C05489=1180.619,-50.249,-42.680,179.529,5.743,149.159
C05490=1180.625,-50.498,-42.668,179.526,5.742,149.160
C05491=1180.631,-50.748,-42.656,179.523,5.742,149.160
C05492=1180.635,-50.998,-42.645,179.521,5.741,149.161
C05493=1180.641,-51.248,-42.633,179.519,5.741,149.162
C05494=1180.645,-51.497,-42.622,179.516,5.741,149.162
C05495=1180.651,-51.747,-42.610,179.514,5.740,149.163
C05496=1180.656,-51.996,-42.599,179.512,5.740,149.163
C05497=1180.662,-52.246,-42.587,179.509,5.740,149.164
C05498=1180.666,-52.496,-42.576,179.507,5.739,149.165
C05499=1180.672,-52.746,-42.565,179.505,5.739,149.165
C05500=1180.677,-52.995,-42.554,179.502,5.738,149.166
C05501=1180.683,-53.245,-42.542,179.500,5.738,149.166
C05502=1180.687,-53.495,-42.531,179.498,5.738,149.167
C05503=1180.693,-53.745,-42.519,179.495,5.737,149.168
C05504=1180.697,-53.994,-42.507,179.493,5.737,149.168
C05505=1180.704,-54.244,-42.496,179.491,5.737,149.169
C05506=1180.708,-54.493,-42.485,179.488,5.737,149.170
C05507=1180.714,-54.743,-42.473,179.486,5.736,149.170
C05508=1180.718,-54.993,-42.461,179.483,5.735,149.171
C05509=1180.723,-55.243,-42.451,179.481,5.736,149.172
C05510=1180.729,-55.492,-42.439,179.479,5.735,149.172
C05511=1180.734,-55.742,-42.428,179.476,5.734,149.173
C05512=1180.739,-55.992,-42.416,179.474,5.735,149.174
C05513=1180.744,-56.242,-42.405,179.472,5.734,149.174
C05514=1180.750,-56.491,-42.393,179.469,5.734,149.175
C05515=1180.755,-56.740,-42.382,179.467,5.733,149.175
C05516=1180.760,-56.991,-42.372,179.465,5.733,149.176
C05517=1180.765,-57.241,-42.360,179.462,5.733,149.177
C05518=1180.771,-57.489,-42.349,179.460,5.732,149.177
C05519=1180.776,-57.739,-42.337,179.458,5.732,149.178
C05520=1180.781,-57.989,-42.326,179.456,5.732,149.179
C05521=1180.786,-58.239,-42.315,179.453,5.731,149.179
C05522=1180.792,-58.489,-42.303,179.451,5.731,149.180
C05523=1180.796,-58.738,-42.292,179.449,5.731,149.180
C05524=1180.802,-58.988,-42.280,179.446,5.731,149.181
C05525=1180.807,-59.238,-42.270,179.444,5.730,149.182
C05526=1180.812,-59.487,-42.259,179.442,5.730,149.182
C05527=1180.818,-59.737,-42.247,179.439,5.730,149.183
C05528=1180.822,-59.987,-42.236,179.437,5.729,149.183
C05529=1180.828,-60.236,-42.225,179.434,5.729,149.184
C05530=1180.833,-60.486,-42.213,179.432,5.729,149.185
C05531=1180.838,-60.736,-42.202,179.430,5.728,149.185
C05532=1180.844,-60.985,-42.192,179.427,5.728,149.186
C05533=1180.849,-61.235,-42.180,179.425,5.728,149.187
C05534=1180.854,-61.485,-42.169,179.423,5.727,149.187
C05535=1180.859,-61.735,-42.159,179.420,5.727,149.188
C05536=1180.865,-61.985,-42.147,179.418,5.727,149.189
C05537=1180.869,-62.234,-42.135,179.416,5.726,149.189
C05538=1180.875,-62.484,-42.125,179.413,5.726,149.190
C05539=1180.880,-62.734,-42.113,179.411,5.725,149.190
C05540=1180.885,-62.983,-42.102,179.409,5.726,149.191
C05541=1180.891,-63.233,-42.092,179.406,5.725,149.192
C05542=1180.895,-63.482,-42.081,179.404,5.724,149.192
C05543=1180.901,-63.732,-42.069,179.402,5.725,149.193
C05544=1180.906,-63.982,-42.058,179.399,5.724,149.194
C05545=1180.911,-64.232,-42.047,179.397,5.723,149.194
C05546=1180.916,-64.482,-42.037,179.395,5.724,149.195
C05547=1180.922,-64.731,-42.025,179.393,5.723,149.196
C05548=1180.927,-64.981,-42.014,179.390,5.723,149.196
C05549=1180.933,-65.230,-42.004,179.388,5.723,149.197
C05550=1180.937,-65.480,-41.992,179.386,5.723,149.197
C05551=1180.943,-65.730,-41.981,179.383,5.722,149.198
C05552=1180.948,-65.979,-41.970,179.381,5.722,149.199
C05553=1180.953,-66.230,-41.960,179.379,5.722,149.199
C05554=1180.959,-66.478,-41.949,179.376,5.721,149.200
C05555=1180.964,-66.729,-41.938,179.374,5.721,149.200
C05556=1180.969,-66.979,-41.926,179.372,5.721,149.201
C05557=1180.974,-67.228,-41.915,179.370,5.720,149.202
C05558=1180.979,-67.478,-41.905,179.367,5.720,149.202
C05559=1180.985,-67.727,-41.894,179.365,5.720,149.203
C05560=1180.990,-67.977,-41.883,179.363,5.719,149.204
C05561=1180.995,-68.227,-41.871,179.360,5.719,149.204
C05562=1181.001,-68.476,-41.861,179.358,5.719,149.205
C05563=1181.006,-68.727,-41.851,179.356,5.718,149.205
C05564=1181.011,-68.976,-41.840,179.353,5.718,149.206
C05565=1181.017,-69.226,-41.828,179.351,5.718,149.207
C05566=1181.022,-69.475,-41.818,179.349,5.718,149.207
C05567=1181.027,-69.725,-41.807,179.346,5.717,149.208
C05568=1181.032,-69.975,-41.796,179.344,5.717,149.209
C05569=1181.037,-70.225,-41.785,179.342,5.717,149.209
C05570=1181.042,-70.474,-41.774,179.340,5.716,149.210
C05571=1181.047,-70.724,-41.764,179.338,5.716,149.210
C05572=1181.053,-70.974,-41.753,179.335,5.716,149.211
C05573=1181.058,-71.223,-41.742,179.333,5.715,149.212
C05574=1181.063,-71.473,-41.731,179.331,5.716,149.212
C05575=1181.069,-71.722,-41.720,179.328,5.715,149.213
C05576=1181.074,-71.973,-41.710,179.326,5.714,149.214
C05577=1181.079,-72.222,-41.700,179.324,5.715,149.214
C05578=1181.084,-72.472,-41.688,179.321,5.714,149.215
C05579=1181.090,-72.721,-41.678,179.319,5.714,149.215
C05580=1181.095,-72.972,-41.668,179.317,5.714,149.216
C05581=1181.101,-73.221,-41.656,179.315,5.713,149.217
C05582=1181.106,-73.471,-41.645,179.312,5.713,149.217
C05583=1181.111,-73.721,-41.635,179.310,5.713,149.218
C05584=1181.116,-73.970,-41.624,179.308,5.712,149.218
C05585=1181.122,-74.220,-41.614,179.306,5.713,149.219
C05586=1181.127,-74.470,-41.603,179.303,5.712,149.220
C05587=1181.132,-74.719,-41.592,179.301,5.711,149.220
C05588=1181.137,-74.969,-41.582,179.299,5.712,149.221
C05589=1181.142,-75.219,-41.571,179.296,5.711,149.222
C05590=1181.148,-75.490,-41.559,179.294,5.711,149.222
C05591=1181.153,-75.761,-41.548,179.291,5.710,149.223
C05592=1181.159,-76.031,-41.536,179.289,5.711,149.224
C05593=1181.165,-76.303,-41.525,179.286,5.710,149.224
C05594=1181.170,-76.553,-41.514,179.284,5.709,149.225
C05595=1181.176,-76.803,-41.504,179.282,5.710,149.226
C05596=1181.181,-77.052,-41.493,179.279,5.709,149.226
C05597=1181.186,-77.302,-41.483,179.277,5.709,149.227
C05598=1181.192,-77.551,-41.472,179.275,5.709,149.227
C05599=1181.197,-77.802,-41.462,179.273,5.708,149.228
C05600=1181.202,-78.051,-41.451,179.270,5.708,149.229
C05601=1181.207,-78.301,-41.440,179.268,5.708,149.229
C05602=1181.213,-78.550,-41.430,179.266,5.707,149.230
C05603=1181.218,-78.801,-41.419,179.263,5.707,149.231
C05604=1181.223,-79.050,-41.409,179.262,5.707,149.231
C05605=1181.229,-79.299,-41.398,179.259,5.707,149.232
C05606=1181.234,-79.549,-41.388,179.257,5.707,149.232
C05607=1181.239,-79.798,-41.378,179.255,5.706,149.233
C05608=1181.244,-80.049,-41.368,179.252,5.706,149.234
C05609=1181.249,-80.298,-41.357,179.251,5.706,149.234
C05610=1181.255,-80.548,-41.347,179.248,5.705,149.235
C05611=1181.260,-80.798,-41.337,179.245,5.705,149.236
C05612=1181.265,-81.047,-41.326,179.244,5.705,149.236
C05613=1181.270,-81.297,-41.315,179.241,5.705,149.237
C05614=1181.276,-81.547,-41.305,179.239,5.705,149.237
C05615=1181.281,-81.797,-41.294,179.237,5.704,149.238
C05616=1181.286,-82.047,-41.284,179.234,5.704,149.239
C05617=1181.292,-82.296,-41.274,179.232,5.704,149.239
C05618=1181.297,-82.546,-41.263,179.230,5.703,149.240
C05619=1181.302,-82.796,-41.254,179.227,5.703,149.241
C05620=1181.307,-83.045,-41.243,179.225,5.703,149.241
C05621=1181.312,-83.295,-41.233,179.223,5.703,149.242
C05622=1181.318,-83.545,-41.223,179.221,5.703,149.242
C05623=1181.323,-83.795,-41.211,179.218,5.702,149.243
C05624=1181.328,-84.044,-41.201,179.216,5.702,149.244
C05625=1181.334,-84.294,-41.191,179.214,5.702,149.244
C05626=1181.339,-84.544,-41.180,179.212,5.701,149.245
C05627=1181.344,-84.793,-41.171,179.210,5.701,149.245
C05628=1181.349,-85.043,-41.161,179.207,5.701,149.246
C05629=1181.354,-85.293,-41.150,179.205,5.700,149.247
C05630=1181.360,-85.542,-41.140,179.203,5.701,149.247
C05631=1181.365,-85.792,-41.130,179.200,5.700,149.248
C05632=1181.370,-86.042,-41.119,179.199,5.700,149.248
C05633=1181.375,-86.291,-41.109,179.196,5.700,149.249
C05634=1181.381,-86.541,-41.099,179.194,5.699,149.250
C05635=1181.386,-86.791,-41.089,179.192,5.699,149.250
C05636=1181.391,-87.041,-41.078,179.189,5.699,149.251
C05637=1181.397,-87.290,-41.068,179.188,5.699,149.252
C05638=1181.402,-87.541,-41.059,179.185,5.699,149.252
C05639=1181.407,-87.790,-41.049,179.183,5.698,149.253
C05640=1181.413,-88.040,-41.039,179.181,5.698,149.253
C05641=1181.418,-88.290,-41.028,179.178,5.698,149.254
C05642=1181.423,-88.539,-41.018,179.176,5.698,149.255
C05643=1181.428,-88.789,-41.008,179.174,5.697,149.255
C05644=1181.433,-89.039,-40.998,179.171,5.697,149.256
C05645=1181.439,-89.289,-40.987,179.169,5.697,149.257
C05646=1181.444,-89.538,-40.977,179.167,5.696,149.257
C05647=1181.449,-89.788,-40.967,179.165,5.697,149.258
C05648=1181.454,-90.038,-40.957,179.162,5.696,149.258
C05649=1181.460,-90.288,-40.947,179.160,5.695,149.259
C05650=1181.465,-90.537,-40.938,179.158,5.696,149.260
C05651=1181.470,-90.787,-40.927,179.156,5.695,149.260
C05652=1181.476,-91.037,-40.917,179.154,5.695,149.261
C05653=1181.481,-91.287,-40.907,179.152,5.695,149.261
C05654=1181.486,-91.536,-40.897,179.149,5.694,149.262
C05655=1181.491,-91.786,-40.887,179.147,5.695,149.263
C05656=1181.497,-92.036,-40.877,179.145,5.694,149.263
C05657=1181.503,-92.286,-40.867,179.143,5.694,149.264
C05658=1181.507,-92.536,-40.857,179.140,5.693,149.264
C05659=1181.512,-92.785,-40.847,179.138,5.693,149.265
C05660=1181.518,-93.035,-40.837,179.136,5.693,149.266
C05661=1181.523,-93.285,-40.828,179.134,5.693,149.266
C05662=1181.528,-93.535,-40.817,179.131,5.693,149.267
C05663=1181.534,-93.784,-40.807,179.129,5.692,149.267
C05664=1181.539,-94.034,-40.797,179.127,5.693,149.268
C05665=1181.545,-94.284,-40.788,179.125,5.692,149.269
C05666=1181.550,-94.533,-40.778,179.122,5.691,149.269
C05667=1181.554,-94.783,-40.768,179.121,5.691,149.270
C05668=1181.560,-95.033,-40.757,179.118,5.691,149.271
C05669=1181.566,-95.283,-40.748,179.116,5.691,149.271
C05670=1181.571,-95.532,-40.738,179.114,5.691,149.272
C05671=1181.576,-95.782,-40.728,179.112,5.691,149.272
C05672=1181.581,-96.032,-40.718,179.109,5.690,149.273
C05673=1181.587,-96.282,-40.709,179.107,5.690,149.274
C05674=1181.592,-96.531,-40.698,179.105,5.690,149.274
C05675=1181.597,-96.781,-40.689,179.103,5.689,149.275
C05676=1181.603,-97.031,-40.679,179.101,5.689,149.275
C05677=1181.608,-97.281,-40.669,179.098,5.689,149.276
C05678=1181.613,-97.530,-40.659,179.097,5.689,149.277
C05679=1181.619,-97.780,-40.650,179.094,5.689,149.277
C05680=1181.624,-98.030,-40.640,179.091,5.688,149.278
C05681=1181.629,-98.279,-40.630,179.090,5.688,149.278
C05682=1181.634,-98.530,-40.620,179.087,5.688,149.279
C05683=1181.639,-98.779,-40.610,179.085,5.688,149.280
C05684=1181.645,-99.029,-40.600,179.083,5.688,149.280
C05685=1181.650,-99.279,-40.591,179.081,5.688,149.281
C05686=1181.656,-99.528,-40.581,179.078,5.687,149.282
C05687=1181.661,-99.777,-40.571,179.077,5.687,149.282
C05688=1181.666,-100.028,-40.562,179.074,5.687,149.283
C05689=1181.671,-100.278,-40.551,179.072,5.686,149.283
C05690=1181.677,-100.528,-40.542,179.070,5.686,149.284
C05691=1181.682,-100.777,-40.532,179.067,5.686,149.285
C05692=1181.687,-101.026,-40.523,179.066,5.686,149.285
C05693=1181.693,-101.277,-40.513,179.063,5.686,149.286
C05694=1181.698,-101.549,-40.503,179.061,5.686,149.286
C05695=1181.704,-101.820,-40.492,179.059,5.685,149.287
C05696=1181.709,-102.092,-40.482,179.056,5.685,149.288
C05697=1181.716,-102.363,-40.471,179.053,5.684,149.289
C05698=1181.721,-102.613,-40.462,179.052,5.685,149.289
C05699=1181.726,-102.863,-40.452,179.049,5.684,149.290
C05700=1181.731,-103.113,-40.442,179.047,5.684,149.290
C05701=1181.737,-103.363,-40.433,179.045,5.684,149.291
C05702=1181.742,-103.612,-40.423,179.043,5.684,149.291
C05703=1181.748,-103.862,-40.414,179.041,5.683,149.292
C05704=1181.753,-104.111,-40.404,179.039,5.683,149.293
C05705=1181.758,-104.362,-40.394,179.036,5.683,149.293
C05706=1181.763,-104.611,-40.385,179.035,5.683,149.294
C05707=1181.768,-104.861,-40.376,179.032,5.683,149.295
C05708=1181.773,-105.111,-40.365,179.030,5.682,149.295
C05709=1181.779,-105.361,-40.356,179.028,5.682,149.296
C05710=1181.784,-105.610,-40.346,179.026,5.681,149.296
C05711=1181.789,-105.860,-40.337,179.023,5.682,149.297
C05712=1181.795,-106.110,-40.327,179.021,5.681,149.298
C05713=1181.800,-106.360,-40.318,179.019,5.681,149.298
C05714=1181.806,-106.610,-40.309,179.016,5.681,149.299
C05715=1181.811,-106.859,-40.299,179.015,5.681,149.299
C05716=1181.816,-107.109,-40.290,179.012,5.681,149.300
C05717=1181.822,-107.358,-40.280,179.011,5.681,149.300
C05718=1181.827,-107.608,-40.271,179.008,5.680,149.301
C05719=1181.832,-107.858,-40.261,179.006,5.680,149.302
C05720=1181.838,-108.108,-40.252,179.004,5.680,149.302
C05721=1181.843,-108.357,-40.243,179.002,5.680,149.303
C05722=1181.848,-108.607,-40.233,178.999,5.680,149.304
C05723=1181.853,-108.858,-40.224,178.997,5.679,149.304
C05724=1181.859,-109.108,-40.214,178.995,5.679,149.305
C05725=1181.864,-109.357,-40.205,178.993,5.678,149.305
C05726=1181.869,-109.607,-40.196,178.991,5.679,149.306
C05727=1181.874,-109.856,-40.185,178.989,5.678,149.306
C05728=1181.880,-110.106,-40.177,178.987,5.678,149.307
C05729=1181.885,-110.356,-40.168,178.984,5.678,149.308
C05730=1181.890,-110.606,-40.157,178.982,5.678,149.308
C05731=1181.896,-110.855,-40.149,178.980,5.677,149.309
C05732=1181.901,-111.105,-40.140,178.978,5.678,149.310
C05733=1181.906,-111.355,-40.129,178.976,5.677,149.310
C05734=1181.912,-111.605,-40.121,178.974,5.677,149.311
C05735=1181.917,-111.855,-40.112,178.972,5.677,149.311
C05736=1181.923,-112.105,-40.102,178.969,5.677,149.312
C05737=1181.927,-112.354,-40.093,178.967,5.676,149.312
C05738=1181.933,-112.604,-40.084,178.965,5.677,149.313
C05739=1181.939,-112.854,-40.074,178.963,5.676,149.314
C05740=1181.944,-113.104,-40.065,178.961,5.676,149.314
C05741=1181.949,-113.353,-40.056,178.959,5.676,149.315
C05742=1181.954,-113.603,-40.046,178.957,5.676,149.316
C05743=1181.960,-113.853,-40.037,178.954,5.675,149.316
C05744=1181.965,-114.103,-40.028,178.953,5.675,149.317
C05745=1181.970,-114.352,-40.019,178.950,5.675,149.317
C05746=1181.976,-114.602,-40.010,178.949,5.675,149.318
C05747=1181.981,-114.851,-40.001,178.946,5.674,149.318
C05748=1181.986,-115.101,-39.992,178.944,5.674,149.319
C05749=1181.992,-115.351,-39.982,178.942,5.674,149.320
C05750=1181.997,-115.601,-39.973,178.939,5.673,149.320
C05751=1182.002,-115.851,-39.964,178.937,5.674,149.321
C05752=1182.008,-116.100,-39.955,178.935,5.673,149.321
C05753=1182.013,-116.351,-39.945,178.933,5.673,149.322
C05754=1182.019,-116.600,-39.937,178.931,5.673,149.323
C05755=1182.024,-116.850,-39.927,178.929,5.673,149.323
C05756=1182.029,-117.099,-39.918,178.927,5.672,149.324
C05757=1182.034,-117.349,-39.909,178.924,5.673,149.324
C05758=1182.040,-117.599,-39.900,178.922,5.672,149.325
C05759=1182.045,-117.849,-39.891,178.920,5.672,149.326
C05760=1182.050,-118.099,-39.882,178.918,5.671,149.326
C05761=1182.055,-118.348,-39.872,178.916,5.671,149.327
C05762=1182.061,-118.598,-39.864,178.914,5.671,149.327
C05763=1182.067,-118.848,-39.854,178.912,5.671,149.328
C05764=1182.072,-119.098,-39.845,178.909,5.671,149.329
C05765=1182.077,-119.347,-39.836,178.908,5.671,149.329
C05766=1182.082,-119.597,-39.828,178.905,5.670,149.330
C05767=1182.087,-119.847,-39.819,178.904,5.670,149.330
C05768=1182.093,-120.097,-39.809,178.901,5.670,149.331
C05769=1182.098,-120.347,-39.800,178.899,5.670,149.331
C05770=1182.104,-120.597,-39.791,178.897,5.670,149.332
C05771=1182.109,-120.847,-39.782,178.895,5.670,149.333
C05772=1182.114,-121.095,-39.773,178.893,5.669,149.333
C05773=1182.119,-121.345,-39.764,178.891,5.669,149.334
C05774=1182.124,-121.595,-39.755,178.889,5.669,149.334
C05775=1182.130,-121.845,-39.746,178.886,5.669,149.335
C05776=1182.136,-122.095,-39.737,178.885,5.669,149.336
C05777=1182.141,-122.345,-39.728,178.882,5.669,149.336
C05778=1182.146,-122.595,-39.719,178.881,5.669,149.337
C05779=1182.151,-122.845,-39.710,178.878,5.668,149.337
C05780=1182.157,-123.094,-39.702,178.876,5.668,149.338
C05781=1182.162,-123.344,-39.693,178.874,5.668,149.338
C05782=1182.167,-123.593,-39.684,178.872,5.668,149.339
C05783=1182.173,-123.844,-39.674,178.870,5.667,149.340
C05784=1182.178,-124.094,-39.666,178.868,5.668,149.340
C05785=1182.183,-124.343,-39.657,178.866,5.667,149.341
C05786=1182.189,-124.593,-39.648,178.863,5.667,149.342
C05787=1182.194,-124.842,-39.639,178.861,5.666,149.342
C05788=1182.199,-125.092,-39.630,178.860,5.666,149.343
C05789=1182.205,-125.342,-39.621,178.857,5.666,149.343
C05790=1182.210,-125.593,-39.613,178.855,5.666,149.344
C05791=1182.215,-125.842,-39.604,178.853,5.666,149.344
C05792=1182.220,-126.092,-39.595,178.851,5.666,149.345
C05793=1182.226,-126.341,-39.587,178.848,5.665,149.346
C05794=1182.231,-126.591,-39.578,178.847,5.665,149.346
C05795=1182.237,-126.841,-39.569,178.845,5.665,149.347
C05796=1182.242,-127.091,-39.560,178.843,5.665,149.347
C05797=1182.248,-127.341,-39.551,178.840,5.664,149.348
C05798=1181.827,-127.352,-39.591,178.837,5.668,149.350
C05799=1181.821,-127.102,-39.600,178.839,5.668,149.349
C05800=1181.816,-126.853,-39.609,178.841,5.669,149.349
C05801=1181.810,-126.603,-39.618,178.843,5.669,149.348
C05802=1181.805,-126.353,-39.626,178.845,5.669,149.348
C05803=1181.800,-126.103,-39.635,178.847,5.669,149.347
C05804=1181.794,-125.852,-39.644,178.849,5.669,149.346
C05805=1181.789,-125.602,-39.653,178.852,5.669,149.346
C05806=1181.783,-125.353,-39.662,178.853,5.669,149.345
C05807=1181.778,-125.103,-39.670,178.855,5.670,149.345
C05808=1181.773,-124.854,-39.679,178.857,5.670,149.344
C05809=1181.767,-124.604,-39.688,178.860,5.670,149.343
C05810=1181.762,-124.354,-39.697,178.862,5.670,149.343
C05811=1181.757,-124.104,-39.706,178.864,5.671,149.342
C05812=1181.751,-123.855,-39.715,178.866,5.670,149.342
C05813=1181.746,-123.605,-39.723,178.868,5.671,149.341
C05814=1181.741,-123.355,-39.732,178.870,5.671,149.341
C05815=1181.736,-123.105,-39.741,178.872,5.671,149.340
C05816=1181.730,-122.855,-39.751,178.874,5.671,149.339
C05817=1181.725,-122.605,-39.760,178.877,5.672,149.339
C05818=1181.720,-122.356,-39.769,178.878,5.672,149.338
C05819=1181.714,-122.106,-39.777,178.881,5.672,149.337
C05820=1181.709,-121.857,-39.786,178.883,5.672,149.337
C05821=1181.704,-121.607,-39.795,178.885,5.673,149.336
C05822=1181.698,-121.357,-39.804,178.887,5.673,149.336
C05823=1181.693,-121.107,-39.813,178.889,5.673,149.335
C05824=1181.687,-120.857,-39.822,178.891,5.673,149.335
C05825=1181.682,-120.607,-39.831,178.893,5.674,149.334
C05826=1181.677,-120.357,-39.840,178.895,5.673,149.333
C05827=1181.671,-120.108,-39.848,178.898,5.674,149.333
C05828=1181.666,-119.859,-39.858,178.900,5.674,149.332
C05829=1181.661,-119.609,-39.867,178.902,5.674,149.332
C05830=1181.655,-119.359,-39.876,178.903,5.674,149.331
C05831=1181.650,-119.109,-39.885,178.906,5.675,149.330
C05832=1181.645,-118.859,-39.894,178.908,5.675,149.330
C05833=1181.640,-118.609,-39.903,178.910,5.675,149.329
C05834=1181.635,-118.359,-39.912,178.912,5.675,149.329
C05835=1181.629,-118.109,-39.922,178.915,5.675,149.328
C05836=1181.623,-117.859,-39.930,178.916,5.675,149.328
C05837=1181.619,-117.610,-39.940,178.919,5.676,149.327
C05838=1181.613,-117.361,-39.949,178.921,5.676,149.326
C05839=1181.608,-117.111,-39.957,178.923,5.676,149.326
C05840=1181.602,-116.861,-39.967,178.925,5.676,149.325
C05841=1181.597,-116.611,-39.976,178.928,5.677,149.324
C05842=1181.591,-116.361,-39.985,178.929,5.677,149.324
C05843=1181.587,-116.112,-39.994,178.931,5.677,149.323
C05844=1181.581,-115.862,-40.004,178.933,5.677,149.323
C05845=1181.576,-115.612,-40.013,178.936,5.678,149.322
C05846=1181.570,-115.362,-40.022,178.938,5.677,149.322
C05847=1181.565,-115.112,-40.031,178.940,5.678,149.321
C05848=1181.559,-114.862,-40.040,178.942,5.678,149.320
C05849=1181.554,-114.613,-40.050,178.944,5.678,149.320
C05850=1181.549,-114.363,-40.059,178.946,5.678,149.319
C05851=1181.544,-114.113,-40.067,178.948,5.679,149.319
C05852=1181.538,-113.863,-40.077,178.951,5.678,149.318
C05853=1181.533,-113.614,-40.087,178.953,5.679,149.317
C05854=1181.528,-113.364,-40.095,178.955,5.679,149.317
C05855=1181.522,-113.114,-40.105,178.957,5.679,149.316
C05856=1181.517,-112.864,-40.114,178.959,5.679,149.316
C05857=1181.512,-112.615,-40.123,178.961,5.680,149.315
C05858=1181.507,-112.365,-40.132,178.963,5.679,149.314
C05859=1181.501,-112.115,-40.142,178.966,5.680,149.314
C05860=1181.496,-111.865,-40.151,178.968,5.680,149.313
C05861=1181.491,-111.616,-40.160,178.970,5.681,149.313
C05862=1181.485,-111.365,-40.170,178.972,5.680,149.312
C05863=1181.480,-111.116,-40.179,178.974,5.681,149.311
C05864=1181.475,-110.866,-40.188,178.976,5.681,149.311
C05865=1181.469,-110.616,-40.198,178.978,5.681,149.310
C05866=1181.464,-110.366,-40.207,178.981,5.682,149.310
C05867=1181.459,-110.117,-40.216,178.983,5.682,149.309
C05868=1181.453,-109.867,-40.226,178.985,5.682,149.308
C05869=1181.448,-109.617,-40.235,178.987,5.682,149.308
C05870=1181.443,-109.367,-40.245,178.990,5.682,149.307
C05871=1181.437,-109.118,-40.254,178.991,5.682,149.307
C05872=1181.432,-108.868,-40.263,178.993,5.683,149.306
C05873=1181.427,-108.618,-40.273,178.995,5.683,149.305
C05874=1181.422,-108.368,-40.282,178.998,5.683,149.305
C05875=1181.416,-108.119,-40.291,179.000,5.683,149.304
C05876=1181.411,-107.869,-40.301,179.002,5.684,149.304
C05877=1181.406,-107.619,-40.310,179.004,5.684,149.303
C05878=1181.400,-107.370,-40.320,179.007,5.684,149.302
C05879=1181.395,-107.120,-40.329,179.008,5.684,149.302
C05880=1181.390,-106.870,-40.338,179.011,5.684,149.301
C05881=1181.384,-106.620,-40.348,179.013,5.684,149.301
C05882=1181.379,-106.371,-40.357,179.015,5.685,149.300
C05883=1181.373,-106.121,-40.367,179.017,5.685,149.299
C05884=1181.368,-105.871,-40.376,179.020,5.685,149.299
C05885=1181.363,-105.622,-40.386,179.022,5.686,149.298
C05886=1181.358,-105.371,-40.396,179.024,5.685,149.298
C05887=1181.353,-105.122,-40.405,179.026,5.686,149.297
C05888=1181.347,-104.872,-40.415,179.028,5.686,149.296
C05889=1181.342,-104.622,-40.424,179.030,5.687,149.296
C05890=1181.336,-104.372,-40.434,179.032,5.686,149.295
C05891=1181.332,-104.123,-40.443,179.035,5.687,149.295
C05892=1181.326,-103.873,-40.453,179.037,5.687,149.294
C05893=1181.321,-103.624,-40.463,179.039,5.687,149.293
C05894=1181.315,-103.373,-40.472,179.042,5.688,149.293
C05895=1181.310,-103.124,-40.482,179.043,5.688,149.292
C05896=1181.305,-102.873,-40.492,179.046,5.688,149.292
C05897=1181.300,-102.624,-40.501,179.047,5.688,149.291
C05898=1181.294,-102.374,-40.511,179.050,5.688,149.290
C05899=1181.288,-102.102,-40.521,179.052,5.688,149.290
C05900=1181.283,-101.831,-40.531,179.054,5.689,149.289
C05901=1181.277,-101.560,-40.542,179.057,5.689,149.288
C05902=1181.271,-101.287,-40.552,179.059,5.689,149.288
C05903=1181.266,-101.038,-40.562,179.061,5.690,149.287
C05904=1181.260,-100.788,-40.572,179.064,5.690,149.287
C05905=1181.255,-100.539,-40.581,179.066,5.690,149.286
C05906=1181.250,-100.289,-40.591,179.068,5.690,149.285
C05907=1181.245,-100.039,-40.601,179.070,5.690,149.285
C05908=1181.240,-99.789,-40.611,179.073,5.691,149.284
C05909=1181.234,-99.539,-40.620,179.075,5.690,149.283
C05910=1181.229,-99.290,-40.630,179.077,5.691,149.283
C05911=1181.223,-99.040,-40.640,179.079,5.691,149.282
C05912=1181.218,-98.790,-40.649,179.081,5.692,149.282
C05913=1181.213,-98.540,-40.660,179.084,5.692,149.281
C05914=1181.208,-98.290,-40.669,179.085,5.692,149.281
C05915=1181.202,-98.041,-40.679,179.088,5.692,149.280
C05916=1181.197,-97.791,-40.688,179.090,5.692,149.279
C05917=1181.192,-97.541,-40.698,179.092,5.693,149.279
C05918=1181.186,-97.292,-40.708,179.094,5.693,149.278
C05919=1181.182,-97.042,-40.718,179.097,5.693,149.277
C05920=1181.176,-96.792,-40.728,179.099,5.693,149.277
C05921=1181.170,-96.542,-40.738,179.101,5.693,149.276
C05922=1181.165,-96.293,-40.747,179.103,5.694,149.276
C05923=1181.160,-96.043,-40.758,179.105,5.694,149.275
C05924=1181.155,-95.793,-40.767,179.108,5.694,149.274
C05925=1181.150,-95.543,-40.777,179.109,5.694,149.274
C05926=1181.144,-95.294,-40.787,179.112,5.695,149.273
C05927=1181.139,-95.044,-40.796,179.114,5.695,149.273
C05928=1181.133,-94.794,-40.806,179.116,5.695,149.272
C05929=1181.128,-94.544,-40.817,179.119,5.695,149.271
C05930=1181.123,-94.295,-40.827,179.121,5.695,149.271
C05931=1181.117,-94.045,-40.836,179.123,5.696,149.270
C05932=1181.112,-93.795,-40.846,179.125,5.696,149.270
C05933=1181.108,-93.545,-40.856,179.128,5.696,149.269
C05934=1181.102,-93.296,-40.866,179.130,5.697,149.268
C05935=1181.096,-93.045,-40.876,179.132,5.697,149.268
C05936=1181.091,-92.796,-40.886,179.134,5.697,149.267
C05937=1181.086,-92.546,-40.896,179.136,5.697,149.266
C05938=1181.081,-92.296,-40.906,179.139,5.697,149.266
C05939=1181.076,-92.047,-40.916,179.141,5.698,149.265
C05940=1181.070,-91.798,-40.926,179.143,5.698,149.265
C05941=1181.065,-91.547,-40.936,179.145,5.699,149.264
C05942=1181.059,-91.297,-40.946,179.147,5.698,149.263
C05943=1181.054,-91.048,-40.956,179.149,5.699,149.263
C05944=1181.049,-90.798,-40.966,179.152,5.699,149.262
C05945=1181.044,-90.548,-40.977,179.154,5.699,149.261
C05946=1181.039,-90.299,-40.986,179.156,5.700,149.261
C05947=1181.033,-90.049,-40.996,179.158,5.699,149.260
C05948=1181.027,-89.799,-41.006,179.161,5.700,149.260
C05949=1181.022,-89.549,-41.017,179.163,5.700,149.259
C05950=1181.018,-89.300,-41.026,179.165,5.701,149.259
C05951=1181.012,-89.050,-41.036,179.168,5.701,149.258
C05952=1181.007,-88.800,-41.047,179.170,5.700,149.257
C05953=1181.001,-88.550,-41.057,179.172,5.701,149.257
C05954=1180.997,-88.301,-41.067,179.174,5.701,149.256
C05955=1180.992,-88.051,-41.077,179.176,5.702,149.255
C05956=1180.986,-87.801,-41.088,179.179,5.702,149.255
C05957=1180.980,-87.551,-41.097,179.181,5.702,149.254
C05958=1180.975,-87.301,-41.108,179.183,5.702,149.254
C05959=1180.970,-87.052,-41.117,179.185,5.702,149.253
C05960=1180.965,-86.802,-41.127,179.187,5.703,149.252
C05961=1180.960,-86.552,-41.138,179.190,5.703,149.252
C05962=1180.954,-86.302,-41.148,179.192,5.703,149.251
C05963=1180.948,-86.053,-41.158,179.194,5.704,149.250
C05964=1180.944,-85.803,-41.168,179.196,5.703,149.250
C05965=1180.938,-85.553,-41.179,179.199,5.704,149.249
C05966=1180.933,-85.304,-41.189,179.201,5.704,149.249
C05967=1180.928,-85.054,-41.199,179.203,5.704,149.248
C05968=1180.922,-84.804,-41.210,179.206,5.705,149.247
C05969=1180.917,-84.555,-41.220,179.208,5.704,149.247
C05970=1180.912,-84.305,-41.230,179.210,5.705,149.246
C05971=1180.907,-84.055,-41.240,179.212,5.706,149.245
C05972=1180.901,-83.806,-41.250,179.214,5.706,149.245
C05973=1180.896,-83.555,-41.261,179.217,5.706,149.244
C05974=1180.891,-83.306,-41.271,179.219,5.706,149.244
C05975=1180.886,-83.056,-41.282,179.221,5.706,149.243
C05976=1180.880,-82.807,-41.292,179.224,5.707,149.242
C05977=1180.876,-82.557,-41.302,179.225,5.707,149.242
C05978=1180.871,-82.307,-41.313,179.228,5.707,149.241
C05979=1180.865,-82.058,-41.323,179.230,5.708,149.241
C05980=1180.859,-81.808,-41.333,179.232,5.708,149.240
C05981=1180.854,-81.558,-41.344,179.235,5.708,149.239
C05982=1180.849,-81.308,-41.354,179.236,5.708,149.239
C05983=1180.844,-81.058,-41.364,179.239,5.708,149.238
C05984=1180.838,-80.808,-41.375,179.241,5.709,149.238
C05985=1180.833,-80.559,-41.385,179.243,5.709,149.237
C05986=1180.828,-80.309,-41.396,179.246,5.709,149.236
C05987=1180.822,-80.060,-41.406,179.248,5.710,149.236
C05988=1180.817,-79.809,-41.417,179.250,5.710,149.235
C05989=1180.812,-79.560,-41.427,179.253,5.710,149.234
C05990=1180.807,-79.310,-41.437,179.255,5.711,149.234
C05991=1180.802,-79.060,-41.447,179.257,5.711,149.233
C05992=1180.796,-78.812,-41.458,179.260,5.711,149.233
C05993=1180.791,-78.561,-41.469,179.262,5.711,149.232
C05994=1180.786,-78.312,-41.479,179.264,5.711,149.231
C05995=1180.781,-78.061,-41.490,179.266,5.712,149.231
C05996=1180.775,-77.812,-41.500,179.269,5.712,149.230
C05997=1180.771,-77.562,-41.511,179.271,5.713,149.230
C05998=1180.765,-77.313,-41.521,179.273,5.713,149.229
C05999=1180.759,-77.063,-41.532,179.275,5.713,149.228
C06000=1180.754,-76.813,-41.542,179.278,5.713,149.228
C06001=1180.749,-76.563,-41.552,179.280,5.714,149.227
C06002=1180.744,-76.314,-41.564,179.282,5.714,149.226
C06003=1180.738,-76.043,-41.575,179.285,5.714,149.226
C06004=1180.732,-75.772,-41.587,179.287,5.715,149.225
C06005=1180.727,-75.501,-41.598,179.289,5.714,149.224
C06006=1180.720,-75.230,-41.609,179.292,5.715,149.224
C06007=1180.716,-74.980,-41.620,179.294,5.715,149.223
C06008=1180.710,-74.731,-41.631,179.297,5.716,149.222
C06009=1180.705,-74.480,-41.641,179.299,5.715,149.222
C06010=1180.700,-74.231,-41.652,179.301,5.716,149.221
C06011=1180.695,-73.981,-41.663,179.304,5.717,149.221
C06012=1180.689,-73.732,-41.673,179.306,5.716,149.220
C06013=1180.684,-73.482,-41.684,179.308,5.717,149.219
C06014=1180.679,-73.232,-41.694,179.310,5.717,149.219
C06015=1180.674,-72.982,-41.705,179.312,5.717,149.218
C06016=1180.668,-72.733,-41.716,179.315,5.718,149.217
C06017=1180.663,-72.483,-41.727,179.317,5.717,149.217
C06018=1180.657,-72.233,-41.737,179.319,5.718,149.216
C06019=1180.652,-71.984,-41.749,179.322,5.719,149.216
C06020=1180.647,-71.734,-41.759,179.324,5.719,149.215
C06021=1180.642,-71.484,-41.769,179.326,5.719,149.214
C06022=1180.637,-71.234,-41.781,179.329,5.719,149.214
C06023=1180.632,-70.985,-41.791,179.330,5.720,149.213
C06024=1180.627,-70.735,-41.802,179.333,5.720,149.212
C06025=1180.621,-70.485,-41.813,179.336,5.720,149.212
C06026=1180.616,-70.235,-41.824,179.337,5.720,149.211
C06027=1180.610,-69.986,-41.834,179.340,5.721,149.211
C06028=1180.605,-69.736,-41.845,179.343,5.721,149.210
C06029=1180.600,-69.487,-41.856,179.344,5.721,149.209
C06030=1180.595,-69.237,-41.867,179.347,5.722,149.209
C06031=1180.589,-68.987,-41.878,179.349,5.722,149.208
C06032=1180.584,-68.737,-41.889,179.351,5.722,149.208
C06033=1180.579,-68.487,-41.900,179.354,5.722,149.207
C06034=1180.574,-68.238,-41.910,179.356,5.723,149.206
C06035=1180.569,-67.988,-41.921,179.358,5.723,149.206
C06036=1180.563,-67.739,-41.932,179.361,5.723,149.205
C06037=1180.558,-67.488,-41.943,179.363,5.724,149.204
C06038=1180.552,-67.239,-41.954,179.365,5.724,149.204
C06039=1180.547,-66.989,-41.964,179.368,5.724,149.203
C06040=1180.543,-66.739,-41.976,179.370,5.725,149.203
C06041=1180.537,-66.490,-41.986,179.373,5.725,149.202
C06042=1180.532,-66.240,-41.998,179.374,5.725,149.201
C06043=1180.526,-65.991,-42.009,179.377,5.726,149.201
C06044=1180.521,-65.741,-42.019,179.380,5.726,149.200
C06045=1180.517,-65.491,-42.030,179.381,5.726,149.199
C06046=1180.510,-65.241,-42.041,179.384,5.727,149.199
C06047=1180.506,-64.992,-42.053,179.387,5.727,149.198
C06048=1180.501,-64.741,-42.063,179.388,5.727,149.198
C06049=1180.495,-64.492,-42.074,179.391,5.727,149.197
C06050=1180.490,-64.242,-42.086,179.393,5.728,149.196
C06051=1180.484,-63.993,-42.096,179.395,5.728,149.196
C06052=1180.480,-63.743,-42.107,179.398,5.728,149.195
C06053=1180.475,-63.493,-42.118,179.400,5.729,149.195
C06054=1180.469,-63.244,-42.130,179.402,5.729,149.194
C06055=1180.464,-62.994,-42.141,179.405,5.729,149.193
C06056=1180.459,-62.744,-42.151,179.407,5.730,149.193
C06057=1180.453,-62.495,-42.163,179.410,5.730,149.192
C06058=1180.448,-62.245,-42.174,179.412,5.730,149.191
C06059=1180.443,-61.995,-42.185,179.414,5.731,149.191
C06060=1180.438,-61.746,-42.196,179.416,5.731,149.190
C06061=1180.432,-61.496,-42.208,179.419,5.731,149.189
C06062=1180.427,-61.246,-42.218,179.421,5.732,149.189
C06063=1180.422,-60.997,-42.229,179.423,5.732,149.188
C06064=1180.417,-60.747,-42.241,179.425,5.732,149.187
C06065=1180.412,-60.497,-42.252,179.428,5.732,149.187
C06066=1180.406,-60.248,-42.262,179.430,5.733,149.186
C06067=1180.401,-59.998,-42.274,179.433,5.733,149.186
C06068=1180.396,-59.748,-42.285,179.435,5.733,149.185
C06069=1180.391,-59.498,-42.296,179.437,5.734,149.184
C06070=1180.385,-59.249,-42.308,179.440,5.734,149.184
C06071=1180.381,-58.999,-42.319,179.442,5.734,149.183
C06072=1180.375,-58.749,-42.330,179.444,5.735,149.182
C06073=1180.370,-58.500,-42.341,179.447,5.735,149.182
C06074=1180.365,-58.250,-42.352,179.449,5.736,149.181
C06075=1180.359,-58.000,-42.364,179.451,5.735,149.181
C06076=1180.355,-57.750,-42.376,179.453,5.736,149.180
C06077=1180.349,-57.501,-42.386,179.456,5.737,149.179
C06078=1180.344,-57.251,-42.398,179.458,5.736,149.179
C06079=1180.339,-57.001,-42.409,179.460,5.737,149.178
C06080=1180.334,-56.751,-42.421,179.463,5.737,149.178
C06081=1180.328,-56.502,-42.432,179.466,5.738,149.177
C06082=1180.323,-56.252,-42.442,179.467,5.738,149.176
C06083=1180.318,-56.002,-42.454,179.470,5.738,149.176
C06084=1180.313,-55.753,-42.466,179.473,5.739,149.175
C06085=1180.307,-55.503,-42.477,179.474,5.739,149.174
C06086=1180.302,-55.254,-42.488,179.477,5.739,149.174
C06087=1180.297,-55.004,-42.500,179.479,5.740,149.173
C06088=1180.292,-54.754,-42.511,179.482,5.740,149.173
C06089=1180.286,-54.504,-42.522,179.484,5.740,149.172
C06090=1180.281,-54.255,-42.534,179.486,5.740,149.171
C06091=1180.277,-54.005,-42.545,179.489,5.741,149.171
C06092=1180.271,-53.755,-42.557,179.491,5.742,149.170
C06093=1180.267,-53.506,-42.568,179.493,5.741,149.169
C06094=1180.260,-53.256,-42.580,179.495,5.742,149.169
C06095=1180.256,-53.007,-42.591,179.498,5.743,149.168
C06096=1180.250,-52.757,-42.603,179.501,5.743,149.167
C06097=1180.246,-52.507,-42.614,179.502,5.743,149.167
C06098=1180.240,-52.257,-42.626,179.505,5.743,149.166
C06099=1180.235,-52.008,-42.637,179.508,5.744,149.166
C06100=1180.229,-51.758,-42.648,179.509,5.744,149.165
C06101=1180.225,-51.508,-42.659,179.512,5.744,149.164
C06102=1180.219,-51.258,-42.671,179.515,5.745,149.164
C06103=1180.214,-51.009,-42.682,179.517,5.746,149.163
C06104=1180.208,-50.759,-42.694,179.519,5.745,149.162
C06105=1180.203,-50.509,-42.706,179.522,5.746,149.162
C06106=1180.198,-50.260,-42.717,179.524,5.746,149.161
C06107=1180.193,-49.989,-42.730,179.526,5.747,149.161
C06108=1180.187,-49.720,-42.743,179.529,5.747,149.160
C06109=1180.181,-49.449,-42.755,179.532,5.748,149.159
C06110=1180.176,-49.178,-42.768,179.534,5.748,149.158
C06111=1180.170,-48.929,-42.779,179.537,5.748,149.158
C06112=1180.165,-48.680,-42.791,179.539,5.749,149.157
C06113=1180.160,-48.430,-42.803,179.541,5.749,149.157
C06114=1180.155,-48.180,-42.814,179.544,5.749,149.156
C06115=1180.150,-47.930,-42.826,179.546,5.749,149.155
C06116=1180.144,-47.680,-42.838,179.548,5.750,149.155
C06117=1180.140,-47.430,-42.849,179.551,5.750,149.154
C06118=1180.134,-47.181,-42.861,179.553,5.751,149.154
C06119=1180.129,-46.932,-42.872,179.555,5.751,149.153
C06120=1180.124,-46.682,-42.884,179.558,5.751,149.152
C06121=1180.118,-46.432,-42.896,179.560,5.752,149.152
C06122=1180.114,-46.183,-42.908,179.563,5.752,149.151
C06123=1180.108,-45.933,-42.919,179.565,5.752,149.150
C06124=1180.103,-45.683,-42.931,179.567,5.753,149.150
C06125=1180.098,-45.433,-42.943,179.570,5.753,149.149
C06126=1180.093,-45.183,-42.955,179.572,5.754,149.148
C06127=1180.087,-44.934,-42.966,179.574,5.755,149.148
C06128=1180.082,-44.685,-42.978,179.577,5.754,149.147
C06129=1180.077,-44.435,-42.990,179.579,5.755,149.146
C06130=1180.071,-44.185,-43.002,179.581,5.755,149.146
C06131=1180.067,-43.936,-43.013,179.584,5.756,149.145
C06132=1180.061,-43.686,-43.025,179.586,5.755,149.145
C06133=1180.056,-43.436,-43.038,179.588,5.756,149.144
C06134=1180.052,-43.187,-43.049,179.591,5.757,149.143
C06135=1180.046,-42.937,-43.061,179.594,5.757,149.143
C06136=1180.041,-42.687,-43.073,179.596,5.758,149.142
C06137=1180.035,-42.437,-43.085,179.598,5.758,149.142
C06138=1180.031,-42.188,-43.097,179.601,5.758,149.141
C06139=1180.025,-41.938,-43.108,179.603,5.758,149.140
C06140=1180.020,-41.688,-43.120,179.605,5.759,149.140
C06141=1180.015,-41.438,-43.132,179.607,5.759,149.139
C06142=1180.010,-41.190,-43.144,179.610,5.759,149.138
C06143=1180.004,-40.940,-43.156,179.612,5.760,149.138
C06144=1179.999,-40.690,-43.168,179.615,5.761,149.137
C06145=1179.994,-40.441,-43.180,179.618,5.761,149.136
C06146=1179.989,-40.191,-43.192,179.619,5.761,149.136
C06147=1179.984,-39.941,-43.203,179.622,5.762,149.135
C06148=1179.978,-39.692,-43.216,179.625,5.762,149.135
C06149=1179.973,-39.442,-43.228,179.627,5.763,149.134
C06150=1179.968,-39.192,-43.239,179.629,5.763,149.133
C06151=1179.963,-38.943,-43.252,179.632,5.763,149.133
C06152=1179.958,-38.693,-43.264,179.634,5.764,149.132
C06153=1179.952,-38.443,-43.276,179.636,5.764,149.131
C06154=1179.947,-38.194,-43.288,179.639,5.765,149.131
C06155=1179.942,-37.944,-43.300,179.641,5.765,149.130
C06156=1179.937,-37.694,-43.311,179.643,5.765,149.130
C06157=1179.932,-37.445,-43.324,179.646,5.765,149.129
C06158=1179.926,-37.195,-43.336,179.648,5.766,149.128
C06159=1179.921,-36.945,-43.348,179.651,5.767,149.128
C06160=1179.916,-36.696,-43.360,179.653,5.767,149.127
C06161=1179.910,-36.446,-43.372,179.656,5.767,149.126
C06162=1179.906,-36.197,-43.384,179.658,5.768,149.126
C06163=1179.901,-35.947,-43.396,179.660,5.768,149.125
C06164=1179.896,-35.697,-43.409,179.663,5.768,149.124
C06165=1179.890,-35.447,-43.421,179.665,5.769,149.124
C06166=1179.886,-35.197,-43.434,179.667,5.769,149.123
C06167=1179.880,-34.947,-43.445,179.670,5.769,149.123
C06168=1179.875,-34.697,-43.457,179.672,5.770,149.122
C06169=1179.870,-34.448,-43.470,179.675,5.771,149.121
C06170=1179.864,-34.198,-43.482,179.677,5.771,149.121
C06171=1179.860,-33.949,-43.494,179.680,5.772,149.120
C06172=1179.854,-33.699,-43.506,179.682,5.772,149.120
C06173=1179.849,-33.450,-43.518,179.684,5.772,149.119
C06174=1179.844,-33.200,-43.530,179.687,5.773,149.118
C06175=1179.839,-32.951,-43.543,179.689,5.773,149.118
C06176=1179.833,-32.701,-43.555,179.692,5.774,149.117
C06177=1179.828,-32.451,-43.567,179.694,5.775,149.117
C06178=1179.823,-32.202,-43.580,179.696,5.774,149.116
C06179=1179.818,-31.952,-43.592,179.699,5.775,149.115
C06180=1179.813,-31.702,-43.605,179.701,5.775,149.114
C06181=1179.808,-31.452,-43.617,179.704,5.776,149.114
C06182=1179.803,-31.203,-43.629,179.706,5.776,149.113
C06183=1179.797,-30.953,-43.641,179.709,5.777,149.113
C06184=1179.792,-30.704,-43.654,179.711,5.777,149.112
C06185=1179.787,-30.454,-43.666,179.713,5.777,149.111
C06186=1179.781,-30.204,-43.678,179.716,5.778,149.111
C06187=1179.776,-29.955,-43.691,179.718,5.778,149.110
C06188=1179.771,-29.705,-43.703,179.721,5.779,149.110
C06189=1179.766,-29.455,-43.716,179.723,5.779,149.109
C06190=1179.761,-29.206,-43.728,179.725,5.779,149.108
C06191=1179.756,-28.956,-43.740,179.728,5.780,149.108
C06192=1179.751,-28.707,-43.753,179.730,5.780,149.107
C06193=1179.746,-28.457,-43.765,179.732,5.781,149.106
C06194=1179.740,-28.207,-43.777,179.735,5.782,149.106
C06195=1179.735,-27.958,-43.790,179.738,5.782,149.105
C06196=1179.730,-27.708,-43.803,179.740,5.782,149.104
C06197=1179.725,-27.458,-43.815,179.742,5.782,149.104
C06198=1179.720,-27.209,-43.827,179.745,5.783,149.103
C06199=1179.715,-26.959,-43.840,179.747,5.783,149.103
C06200=1179.710,-26.710,-43.852,179.750,5.784,149.102
C06201=1179.704,-26.460,-43.864,179.752,5.785,149.101
C06202=1179.700,-26.210,-43.877,179.755,5.785,149.101
C06203=1179.695,-25.961,-43.890,179.756,5.785,149.100
C06204=1179.689,-25.711,-43.902,179.759,5.786,149.100
C06205=1179.684,-25.462,-43.914,179.762,5.786,149.099
C06206=1179.678,-25.212,-43.928,179.764,5.787,149.098
C06207=1179.674,-24.962,-43.941,179.767,5.787,149.098
C06208=1179.669,-24.713,-43.953,179.769,5.788,149.097
C06209=1179.663,-24.463,-43.965,179.772,5.788,149.096
C06210=1179.658,-24.213,-43.978,179.774,5.789,149.096
C06211=1179.653,-23.944,-43.991,179.777,5.789,149.095
C06212=1179.647,-23.674,-44.006,179.779,5.790,149.094
C06213=1179.641,-23.404,-44.018,179.782,5.790,149.094
C06214=1179.636,-23.134,-44.032,179.785,5.791,149.093
C06215=1179.630,-22.885,-44.045,179.787,5.790,149.092
C06216=1179.625,-22.635,-44.058,179.789,5.791,149.092
C06217=1179.621,-22.385,-44.071,179.792,5.792,149.091
C06218=1179.616,-22.136,-44.083,179.794,5.792,149.090
C06219=1179.611,-21.887,-44.096,179.796,5.793,149.090
C06220=1179.604,-21.636,-44.108,179.799,5.793,149.089
C06221=1179.600,-21.386,-44.121,179.802,5.794,149.089
C06222=1179.595,-21.137,-44.134,179.804,5.795,149.088
C06223=1179.590,-20.888,-44.146,179.807,5.795,149.087
C06224=1179.584,-20.638,-44.159,179.809,5.795,149.087
C06225=1179.579,-20.388,-44.173,179.811,5.796,149.086
C06226=1179.574,-20.139,-44.185,179.814,5.796,149.086
C06227=1179.569,-19.889,-44.198,179.816,5.797,149.085
C06228=1179.564,-19.640,-44.210,179.819,5.797,149.084
C06229=1179.559,-19.390,-44.223,179.821,5.798,149.084
C06230=1179.553,-19.140,-44.237,179.824,5.798,149.083
C06231=1179.548,-18.891,-44.249,179.826,5.799,149.082
C06232=1179.544,-18.641,-44.262,179.829,5.800,149.082
C06233=1179.538,-18.391,-44.274,179.831,5.799,149.081
C06234=1179.533,-18.142,-44.287,179.833,5.800,149.080
C06235=1179.527,-17.892,-44.300,179.835,5.801,149.080
C06236=1179.523,-17.642,-44.313,179.838,5.801,149.079
C06237=1179.518,-17.393,-44.325,179.841,5.801,149.079
C06238=1179.512,-17.143,-44.339,179.843,5.802,149.078
C06239=1179.508,-16.894,-44.352,179.846,5.803,149.077
C06240=1179.503,-16.645,-44.365,179.848,5.803,149.077
C06241=1179.497,-16.395,-44.378,179.850,5.804,149.076
C06242=1179.492,-16.145,-44.391,179.853,5.804,149.076
C06243=1179.487,-15.896,-44.404,179.855,5.804,149.075
C06244=1179.481,-15.646,-44.417,179.858,5.805,149.074
C06245=1179.477,-15.396,-44.430,179.860,5.805,149.074
C06246=1179.472,-15.147,-44.442,179.863,5.806,149.073
C06247=1179.466,-14.897,-44.456,179.865,5.806,149.072
C06248=1179.461,-14.647,-44.469,179.867,5.807,149.072
C06249=1179.456,-14.398,-44.481,179.870,5.808,149.071
C06250=1179.450,-14.148,-44.494,179.873,5.808,149.070
C06251=1179.446,-13.898,-44.507,179.875,5.809,149.070
C06252=1179.441,-13.649,-44.521,179.878,5.809,149.069
C06253=1179.436,-13.399,-44.534,179.880,5.810,149.069
C06254=1179.430,-13.150,-44.547,179.882,5.811,149.068
C06255=1179.425,-12.900,-44.559,179.885,5.810,149.067
C06256=1179.420,-12.650,-44.573,179.887,5.811,149.067
C06257=1179.415,-12.401,-44.586,179.890,5.811,149.066
C06258=1179.409,-12.152,-44.599,179.892,5.812,149.066
C06259=1179.405,-11.902,-44.612,179.895,5.813,149.065
C06260=1179.400,-11.652,-44.625,179.897,5.813,149.064
C06261=1179.394,-11.402,-44.639,179.899,5.814,149.064
C06262=1179.389,-11.153,-44.651,179.902,5.814,149.063
C06263=1179.384,-10.904,-44.665,179.905,5.815,149.062
C06264=1179.379,-10.654,-44.678,179.907,5.816,149.062
C06265=1179.374,-10.404,-44.691,179.910,5.816,149.061
C06266=1179.369,-10.154,-44.704,179.912,5.816,149.061
C06267=1179.364,-9.905,-44.717,179.914,5.817,149.060
C06268=1179.359,-9.655,-44.731,179.917,5.818,149.059
C06269=1179.354,-9.406,-44.744,179.919,5.817,149.059
C06270=1179.348,-9.156,-44.757,179.921,5.818,149.058
C06271=1179.344,-8.907,-44.771,179.924,5.819,149.058
C06272=1179.338,-8.657,-44.784,179.927,5.819,149.057
C06273=1179.333,-8.407,-44.797,179.929,5.820,149.056
C06274=1179.328,-8.158,-44.809,179.932,5.820,149.056
C06275=1179.323,-7.908,-44.824,179.934,5.821,149.055
C06276=1179.318,-7.659,-44.836,179.937,5.821,149.054
C06277=1179.313,-7.408,-44.850,179.939,5.822,149.054
C06278=1179.308,-7.160,-44.863,179.942,5.823,149.053
C06279=1179.303,-6.909,-44.877,179.944,5.823,149.052
C06280=1179.298,-6.660,-44.889,179.946,5.824,149.052
C06281=1179.293,-6.410,-44.904,179.949,5.824,149.051
C06282=1179.287,-6.161,-44.917,179.952,5.825,149.051
C06283=1179.283,-5.911,-44.930,179.954,5.826,149.050
C06284=1179.277,-5.662,-44.944,179.957,5.826,149.049
C06285=1179.272,-5.412,-44.956,179.959,5.827,149.049
C06286=1179.267,-5.163,-44.971,179.961,5.828,149.048
C06287=1179.261,-4.913,-44.983,179.964,5.828,149.048
C06288=1179.257,-4.664,-44.997,179.967,5.828,149.047
C06289=1179.252,-4.414,-45.010,179.969,5.829,149.046
C06290=1179.246,-4.164,-45.024,179.972,5.830,149.046
C06291=1179.241,-3.914,-45.038,179.974,5.830,149.045
C06292=1179.236,-3.665,-45.050,179.976,5.830,149.044
C06293=1179.231,-3.415,-45.065,179.978,5.831,149.044
C06294=1179.226,-3.166,-45.077,179.981,5.831,149.043
C06295=1179.221,-2.916,-45.092,179.984,5.832,149.043
C06296=1179.215,-2.667,-45.105,179.986,5.833,149.042
C06297=1179.211,-2.417,-45.118,179.989,5.833,149.041
C06298=1179.205,-2.168,-45.132,179.991,5.833,149.041
C06299=1179.201,-1.918,-45.145,179.993,5.834,149.040
C06300=1179.195,-1.668,-45.159,179.996,5.835,149.040
C06301=1179.190,-1.419,-45.173,179.999,5.835,149.039
C06302=1179.185,-1.169,-45.185,-179.999,5.836,149.038
C06303=1179.180,-0.920,-45.200,-179.996,5.837,149.038
C06304=1179.175,-0.669,-45.213,-179.994,5.837,149.037
C06305=1179.170,-0.421,-45.227,-179.992,5.838,149.037
C06306=1179.165,-0.171,-45.241,-179.989,5.838,149.036
C06307=1179.159,0.079,-45.254,-179.986,5.839,149.035
C06308=1179.155,0.328,-45.268,-179.984,5.840,149.035
C06309=1179.149,0.578,-45.281,-179.981,5.840,149.034
C06310=1179.144,0.827,-45.295,-179.979,5.841,149.033
C06311=1179.140,1.077,-45.308,-179.976,5.841,149.033
C06312=1179.134,1.326,-45.322,-179.974,5.842,149.032
C06313=1179.129,1.576,-45.336,-179.971,5.842,149.032
C06314=1179.123,1.826,-45.350,-179.969,5.843,149.031
C06315=1179.118,2.095,-45.364,-179.967,5.844,149.030
C06316=1179.113,2.364,-45.379,-179.964,5.844,149.030
C06317=1179.108,2.634,-45.394,-179.961,5.845,149.029
C06318=1179.102,2.903,-45.409,-179.958,5.846,149.028
C06319=1179.097,3.152,-45.423,-179.955,5.846,149.028
C06320=1179.092,3.402,-45.437,-179.953,5.847,149.027
C06321=1179.087,3.651,-45.450,-179.950,5.848,149.026
C06322=1179.082,3.901,-45.464,-179.948,5.848,149.026
C06323=1179.077,4.151,-45.478,-179.945,5.849,149.025
C06324=1179.071,4.400,-45.491,-179.943,5.849,149.025
C06325=1179.067,4.650,-45.505,-179.940,5.850,149.024
C06326=1179.062,4.899,-45.519,-179.938,5.850,149.023
C06327=1179.056,5.148,-45.533,-179.936,5.851,149.023
C06328=1179.051,5.399,-45.547,-179.933,5.852,149.022
C06329=1179.046,5.648,-45.561,-179.930,5.852,149.021
C06330=1179.041,5.897,-45.575,-179.928,5.853,149.021
C06331=1179.036,6.147,-45.589,-179.925,5.853,149.020
C06332=1179.031,6.397,-45.602,-179.923,5.854,149.020
C06333=1179.025,6.646,-45.616,-179.921,5.855,149.019
C06334=1179.020,6.896,-45.631,-179.918,5.855,149.018
C06335=1179.016,7.145,-45.644,-179.915,5.856,149.018
C06336=1179.010,7.394,-45.658,-179.913,5.857,149.017
C06337=1179.006,7.644,-45.672,-179.910,5.857,149.017
C06338=1179.000,7.894,-45.686,-179.908,5.858,149.016
C06339=1178.995,8.143,-45.700,-179.906,5.858,149.015
C06340=1178.990,8.393,-45.714,-179.903,5.859,149.015
C06341=1178.985,8.643,-45.728,-179.900,5.859,149.014
C06342=1178.980,8.892,-45.743,-179.898,5.860,149.014
C06343=1178.975,9.141,-45.756,-179.896,5.861,149.013
C06344=1178.970,9.391,-45.770,-179.893,5.861,149.012
C06345=1178.965,9.641,-45.784,-179.891,5.862,149.012
C06346=1178.960,9.891,-45.798,-179.888,5.862,149.011
C06347=1178.954,10.140,-45.812,-179.885,5.863,149.010
C06348=1178.949,10.390,-45.826,-179.883,5.865,149.010
C06349=1178.944,10.639,-45.841,-179.880,5.865,149.009
C06350=1178.939,10.888,-45.855,-179.877,5.866,149.009
C06351=1178.934,11.138,-45.869,-179.875,5.866,149.008
C06352=1178.929,11.388,-45.883,-179.873,5.867,149.007
C06353=1178.924,11.637,-45.897,-179.870,5.867,149.007
C06354=1178.919,11.887,-45.912,-179.868,5.868,149.006
C06355=1178.913,12.136,-45.926,-179.865,5.869,149.006
C06356=1178.909,12.386,-45.939,-179.862,5.869,149.005
C06357=1178.904,12.635,-45.953,-179.860,5.870,149.005
C06358=1178.899,12.885,-45.968,-179.858,5.871,149.004
C06359=1178.894,13.134,-45.982,-179.855,5.871,149.003
C06360=1178.889,13.384,-45.996,-179.853,5.872,149.003
C06361=1178.884,13.633,-46.010,-179.850,5.872,149.002
C06362=1178.879,13.883,-46.025,-179.847,5.873,149.001
C06363=1178.874,14.133,-46.039,-179.845,5.874,149.001
C06364=1178.868,14.382,-46.053,-179.843,5.874,149.000
C06365=1178.863,14.632,-46.067,-179.840,5.875,148.999
C06366=1178.858,14.881,-46.081,-179.837,5.876,148.999
C06367=1178.854,15.131,-46.096,-179.835,5.877,148.998
C06368=1178.848,15.381,-46.110,-179.832,5.877,148.998
C06369=1178.842,15.630,-46.124,-179.830,5.878,148.997
C06370=1178.837,15.880,-46.139,-179.827,5.879,148.997
C06371=1178.833,16.129,-46.154,-179.824,5.879,148.996
C06372=1178.828,16.378,-46.168,-179.822,5.880,148.995
C06373=1178.823,16.628,-46.182,-179.820,5.880,148.995
C06374=1178.818,16.878,-46.196,-179.817,5.881,148.994
C06375=1178.812,17.127,-46.210,-179.815,5.882,148.994
C06376=1178.807,17.377,-46.225,-179.812,5.882,148.993
C06377=1178.802,17.626,-46.239,-179.810,5.883,148.992
C06378=1178.798,17.875,-46.254,-179.807,5.884,148.992
C06379=1178.793,18.125,-46.268,-179.804,5.885,148.991
C06380=1178.788,18.375,-46.282,-179.802,5.885,148.990
C06381=1178.783,18.625,-46.297,-179.799,5.886,148.990
C06382=1178.777,18.874,-46.311,-179.797,5.887,148.989
C06383=1178.772,19.123,-46.326,-179.794,5.887,148.989
C06384=1178.767,19.373,-46.340,-179.792,5.888,148.988
C06385=1178.762,19.622,-46.355,-179.789,5.888,148.987
C06386=1178.757,19.872,-46.369,-179.787,5.889,148.987
C06387=1178.752,20.121,-46.384,-179.784,5.890,148.986
C06388=1178.747,20.371,-46.398,-179.782,5.890,148.986
C06389=1178.742,20.621,-46.413,-179.779,5.892,148.985
C06390=1178.737,20.871,-46.427,-179.776,5.892,148.984
C06391=1178.732,21.119,-46.442,-179.774,5.893,148.984
C06392=1178.727,21.369,-46.456,-179.772,5.894,148.983
C06393=1178.722,21.618,-46.471,-179.769,5.894,148.983
C06394=1178.716,21.868,-46.486,-179.766,5.895,148.982
C06395=1178.711,22.118,-46.501,-179.764,5.896,148.982
C06396=1178.706,22.367,-46.515,-179.761,5.896,148.981
C06397=1178.702,22.616,-46.530,-179.759,5.897,148.980
C06398=1178.697,22.866,-46.544,-179.757,5.897,148.980
C06399=1178.691,23.116,-46.559,-179.753,5.899,148.979
C06400=1178.686,23.365,-46.574,-179.751,5.899,148.978
C06401=1178.681,23.615,-46.588,-179.749,5.900,148.978
C06402=1178.676,23.865,-46.602,-179.746,5.901,148.977
C06403=1178.672,24.114,-46.617,-179.743,5.901,148.977
C06404=1178.666,24.364,-46.632,-179.741,5.902,148.976
C06405=1178.661,24.613,-46.647,-179.739,5.902,148.975
C06406=1178.657,24.863,-46.662,-179.736,5.903,148.975
C06407=1178.651,25.113,-46.676,-179.733,5.905,148.974
C06408=1178.646,25.362,-46.691,-179.730,5.905,148.974
C06409=1178.641,25.611,-46.706,-179.728,5.906,148.973
C06410=1178.637,25.860,-46.721,-179.726,5.906,148.972
C06411=1178.631,26.110,-46.736,-179.723,5.907,148.972
C06412=1178.626,26.360,-46.751,-179.721,5.908,148.971
C06413=1178.621,26.609,-46.765,-179.718,5.908,148.971
C06414=1178.616,26.859,-46.780,-179.716,5.909,148.970
C06415=1178.611,27.108,-46.795,-179.713,5.910,148.970
C06416=1178.606,27.357,-46.810,-179.710,5.911,148.969
C06417=1178.601,27.607,-46.825,-179.708,5.911,148.968
C06418=1178.596,27.857,-46.840,-179.705,5.912,148.968
C06419=1178.591,28.125,-46.855,-179.703,5.913,148.967
C06420=1178.584,28.394,-46.871,-179.699,5.914,148.966
C06421=1178.579,28.663,-46.887,-179.697,5.915,148.966
C06422=1178.573,28.932,-46.903,-179.694,5.915,148.965
C06423=1178.569,29.181,-46.918,-179.692,5.916,148.965
C06424=1178.564,29.431,-46.933,-179.689,5.917,148.964
C06425=1178.559,29.681,-46.948,-179.687,5.918,148.963
C06426=1178.554,29.930,-46.963,-179.684,5.919,148.963
C06427=1178.549,30.180,-46.978,-179.681,5.919,148.962
C06428=1178.544,30.429,-46.993,-179.679,5.920,148.962
C06429=1178.539,30.678,-47.008,-179.677,5.920,148.961
C06430=1178.534,30.928,-47.023,-179.673,5.922,148.960
C06431=1178.529,31.178,-47.037,-179.671,5.923,148.960
C06432=1178.523,31.427,-47.053,-179.669,5.923,148.959
C06433=1178.519,31.676,-47.068,-179.666,5.924,148.959
C06434=1178.514,31.926,-47.082,-179.664,5.924,148.958
C06435=1178.508,32.175,-47.098,-179.661,5.925,148.957
C06436=1178.504,32.424,-47.113,-179.658,5.927,148.957
C06437=1178.498,32.674,-47.128,-179.656,5.927,148.956
C06438=1178.494,32.924,-47.143,-179.653,5.928,148.956
C06439=1178.489,33.174,-47.159,-179.651,5.928,148.955
C06440=1178.484,33.423,-47.173,-179.648,5.929,148.954
C06441=1178.478,33.673,-47.189,-179.646,5.930,148.954
C06442=1178.474,33.922,-47.204,-179.643,5.931,148.953
C06443=1178.468,34.171,-47.219,-179.640,5.932,148.953
C06444=1178.463,34.421,-47.233,-179.638,5.932,148.952
C06445=1178.458,34.670,-47.249,-179.635,5.933,148.952
C06446=1178.453,34.919,-47.264,-179.633,5.933,148.951
C06447=1178.448,35.169,-47.280,-179.631,5.934,148.950
C06448=1178.443,35.419,-47.294,-179.627,5.936,148.950
C06449=1178.438,35.669,-47.310,-179.625,5.936,148.949
C06450=1178.433,35.918,-47.325,-179.623,5.937,148.949
C06451=1178.428,36.167,-47.340,-179.620,5.937,148.948
C06452=1178.423,36.416,-47.355,-179.618,5.938,148.947
C06453=1178.418,36.666,-47.371,-179.615,5.940,148.947
C06454=1178.414,36.916,-47.386,-179.612,5.940,148.946
C06455=1178.408,37.165,-47.401,-179.610,5.941,148.946
C06456=1178.403,37.415,-47.417,-179.607,5.941,148.945
C06457=1178.398,37.664,-47.432,-179.605,5.942,148.945
C06458=1178.393,37.913,-47.447,-179.602,5.944,148.944
C06459=1178.389,38.163,-47.463,-179.599,5.944,148.943
C06460=1178.383,38.412,-47.478,-179.597,5.945,148.943
C06461=1178.378,38.662,-47.493,-179.594,5.946,148.942
C06462=1178.373,38.912,-47.508,-179.592,5.946,148.942
C06463=1178.368,39.161,-47.524,-179.589,5.948,148.941
C06464=1178.363,39.410,-47.539,-179.586,5.948,148.940
C06465=1178.358,39.660,-47.555,-179.584,5.949,148.940
C06466=1178.353,39.910,-47.570,-179.581,5.950,148.939
C06467=1178.348,40.159,-47.585,-179.579,5.950,148.939
C06468=1178.343,40.408,-47.601,-179.576,5.952,148.938
C06469=1178.338,40.658,-47.617,-179.573,5.952,148.937
C06470=1178.333,40.907,-47.632,-179.571,5.953,148.937
C06471=1178.328,41.157,-47.647,-179.569,5.954,148.936
C06472=1178.323,41.406,-47.663,-179.566,5.954,148.936
C06473=1178.318,41.655,-47.678,-179.563,5.956,148.935
C06474=1178.313,41.905,-47.694,-179.561,5.956,148.934
C06475=1178.308,42.155,-47.710,-179.558,5.957,148.934
C06476=1178.303,42.404,-47.725,-179.556,5.958,148.933
C06477=1178.298,42.653,-47.740,-179.553,5.959,148.933
C06478=1178.293,42.903,-47.756,-179.550,5.960,148.932
C06479=1178.288,43.153,-47.772,-179.548,5.960,148.932
C06480=1178.283,43.402,-47.787,-179.546,5.961,148.931
C06481=1178.278,43.652,-47.803,-179.542,5.963,148.930
C06482=1178.273,43.901,-47.818,-179.540,5.963,148.930
C06483=1178.267,44.151,-47.834,-179.538,5.964,148.929
C06484=1178.263,44.399,-47.850,-179.535,5.964,148.929
C06485=1178.258,44.649,-47.865,-179.533,5.965,148.928
C06486=1178.253,44.899,-47.881,-179.530,5.967,148.928
C06487=1178.247,45.148,-47.897,-179.527,5.967,148.927
C06488=1178.243,45.398,-47.912,-179.525,5.968,148.926
C06489=1178.238,45.647,-47.928,-179.522,5.968,148.926
C06490=1178.233,45.897,-47.943,-179.519,5.970,148.925
C06491=1178.228,46.147,-47.959,-179.517,5.971,148.925
C06492=1178.223,46.395,-47.975,-179.515,5.972,148.924
C06493=1178.218,46.645,-47.990,-179.512,5.972,148.924
C06494=1178.213,46.895,-48.006,-179.509,5.973,148.923
C06495=1178.208,47.144,-48.022,-179.507,5.974,148.922
C06496=1178.203,47.393,-48.038,-179.504,5.975,148.922
C06497=1178.198,47.643,-48.054,-179.502,5.976,148.921
C06498=1178.193,47.892,-48.069,-179.499,5.977,148.921
C06499=1178.188,48.141,-48.085,-179.496,5.977,148.920
C06500=1178.183,48.392,-48.101,-179.494,5.978,148.920
C06501=1178.178,48.640,-48.117,-179.491,5.979,148.919
C06502=1178.173,48.890,-48.133,-179.488,5.981,148.918
C06503=1178.168,49.140,-48.149,-179.486,5.981,148.918
C06504=1178.163,49.389,-48.164,-179.484,5.982,148.917
C06505=1178.158,49.638,-48.180,-179.480,5.983,148.917
C06506=1178.153,49.888,-48.196,-179.478,5.984,148.916
C06507=1178.148,50.137,-48.211,-179.476,5.985,148.916
C06508=1178.144,50.387,-48.228,-179.473,5.985,148.915
C06509=1178.138,50.636,-48.244,-179.470,5.987,148.914
C06510=1178.133,50.886,-48.259,-179.468,5.987,148.914
C06511=1178.128,51.135,-48.276,-179.465,5.988,148.913
C06512=1178.123,51.384,-48.292,-179.463,5.989,148.913
C06513=1178.118,51.635,-48.308,-179.460,5.990,148.912
C06514=1178.113,51.883,-48.324,-179.457,5.991,148.912
C06515=1178.108,52.132,-48.339,-179.455,5.991,148.911
C06516=1178.104,52.382,-48.355,-179.452,5.993,148.910
C06517=1178.099,52.631,-48.371,-179.449,5.994,148.910
C06518=1178.094,52.881,-48.387,-179.447,5.994,148.909
C06519=1178.089,53.130,-48.403,-179.445,5.995,148.909
C06520=1178.084,53.380,-48.419,-179.441,5.996,148.908
C06521=1178.079,53.629,-48.436,-179.439,5.997,148.908
C06522=1178.073,53.878,-48.451,-179.437,5.998,148.907
C06523=1178.069,54.148,-48.469,-179.433,5.999,148.906
C06524=1178.063,54.415,-48.486,-179.431,6.000,148.906
C06525=1178.058,54.684,-48.503,-179.428,6.001,148.905
C06526=1178.053,54.953,-48.521,-179.425,6.002,148.904
C06527=1178.047,55.202,-48.538,-179.423,6.003,148.904
C06528=1178.042,55.452,-48.554,-179.420,6.004,148.903
C06529=1178.037,55.701,-48.570,-179.417,6.004,148.903
C06530=1178.032,55.951,-48.585,-179.415,6.005,148.902
C06531=1178.027,56.200,-48.602,-179.412,6.007,148.902
C06532=1178.022,56.449,-48.618,-179.410,6.008,148.901
C06533=1178.017,56.699,-48.634,-179.407,6.008,148.900
C06534=1178.012,56.948,-48.650,-179.404,6.010,148.900
C06535=1178.007,57.198,-48.667,-179.402,6.010,148.899
C06536=1178.002,57.447,-48.682,-179.400,6.011,148.899
C06537=1177.998,57.697,-48.699,-179.396,6.012,148.898
C06538=1177.993,57.945,-48.715,-179.394,6.013,148.898
C06539=1177.988,58.196,-48.731,-179.392,6.014,148.897
C06540=1177.983,58.444,-48.747,-179.388,6.015,148.897
C06541=1177.977,58.695,-48.764,-179.386,6.016,148.896
C06542=1177.973,58.944,-48.781,-179.384,6.017,148.895
C06543=1177.968,59.193,-48.797,-179.381,6.018,148.895
C06544=1177.963,59.443,-48.813,-179.378,6.019,148.894
C06545=1177.958,59.692,-48.829,-179.376,6.020,148.894
C06546=1177.953,59.941,-48.846,-179.373,6.021,148.893
C06547=1177.948,60.191,-48.861,-179.371,6.022,148.893
C06548=1177.943,60.441,-48.879,-179.368,6.022,148.892
C06549=1177.938,60.689,-48.895,-179.365,6.024,148.891
C06550=1177.933,60.939,-48.912,-179.363,6.025,148.891
C06551=1177.928,61.188,-48.927,-179.360,6.025,148.890
C06552=1177.923,61.438,-48.944,-179.357,6.027,148.890
C06553=1177.919,61.687,-48.961,-179.355,6.027,148.889
C06554=1177.913,61.937,-48.977,-179.353,6.028,148.889
C06555=1177.908,62.186,-48.993,-179.349,6.030,148.888
C06556=1177.903,62.435,-49.010,-179.347,6.030,148.888
C06557=1177.899,62.685,-49.026,-179.345,6.031,148.887
C06558=1177.894,62.934,-49.043,-179.342,6.033,148.887
C06559=1177.888,63.184,-49.059,-179.339,6.033,148.886
C06560=1177.883,63.433,-49.076,-179.337,6.034,148.886
C06561=1177.878,63.682,-49.092,-179.334,6.035,148.885
C06562=1177.874,63.932,-49.109,-179.331,6.036,148.884
C06563=1177.869,64.181,-49.126,-179.329,6.037,148.884
C06564=1177.863,64.431,-49.142,-179.326,6.038,148.883
C06565=1177.859,64.680,-49.158,-179.324,6.039,148.883
C06566=1177.854,64.930,-49.175,-179.321,6.040,148.882
C06567=1177.848,65.179,-49.192,-179.318,6.041,148.882
C06568=1177.844,65.428,-49.209,-179.316,6.042,148.881
C06569=1177.839,65.677,-49.225,-179.313,6.043,148.880
C06570=1177.834,65.927,-49.242,-179.310,6.044,148.880
C06571=1177.829,66.176,-49.259,-179.308,6.045,148.879
C06572=1177.824,66.426,-49.275,-179.305,6.046,148.879
C06573=1177.819,66.675,-49.291,-179.303,6.047,148.878
C06574=1177.814,66.925,-49.308,-179.300,6.048,148.878
C06575=1177.809,67.174,-49.325,-179.298,6.049,148.877
C06576=1177.805,67.423,-49.341,-179.295,6.050,148.877
C06577=1177.799,67.673,-49.359,-179.292,6.051,148.876
C06578=1177.795,67.923,-49.375,-179.290,6.052,148.875
C06579=1177.790,68.171,-49.392,-179.287,6.053,148.875
C06580=1177.785,68.421,-49.409,-179.284,6.054,148.874
C06581=1177.780,68.671,-49.426,-179.282,6.055,148.874
C06582=1177.774,68.920,-49.443,-179.279,6.056,148.873
C06583=1177.770,69.169,-49.459,-179.277,6.057,148.873
C06584=1177.765,69.419,-49.476,-179.274,6.058,148.872
C06585=1177.760,69.668,-49.493,-179.271,6.060,148.872
C06586=1177.755,69.917,-49.509,-179.269,6.060,148.871
C06587=1177.750,70.167,-49.527,-179.267,6.061,148.871
C06588=1177.745,70.417,-49.543,-179.263,6.062,148.870
C06589=1177.740,70.665,-49.560,-179.261,6.063,148.869
C06590=1177.735,70.915,-49.577,-179.258,6.065,148.869
C06591=1177.731,71.164,-49.594,-179.255,6.065,148.868
C06592=1177.726,71.414,-49.612,-179.253,6.066,148.868
C06593=1177.721,71.663,-49.628,-179.250,6.067,148.867
C06594=1177.715,71.912,-49.645,-179.248,6.068,148.867
C06595=1177.711,72.162,-49.662,-179.245,6.070,148.866
C06596=1177.706,72.411,-49.678,-179.242,6.070,148.866
C06597=1177.701,72.661,-49.695,-179.240,6.071,148.865
C06598=1177.696,72.910,-49.712,-179.237,6.073,148.865
C06599=1177.691,73.159,-49.730,-179.234,6.073,148.864
C06600=1177.687,73.409,-49.747,-179.232,6.075,148.863
C06601=1177.681,73.658,-49.764,-179.230,6.076,148.863
C06602=1177.676,73.907,-49.780,-179.226,6.077,148.862
C06603=1177.671,74.157,-49.798,-179.224,6.078,148.862
C06604=1177.667,74.406,-49.815,-179.222,6.079,148.861
C06605=1177.662,74.656,-49.832,-179.219,6.080,148.861
C06606=1177.656,74.905,-49.849,-179.216,6.081,148.860
C06607=1177.651,75.154,-49.866,-179.214,6.082,148.860
C06608=1177.647,75.403,-49.884,-179.211,6.083,148.859
C06609=1177.642,75.653,-49.900,-179.208,6.085,148.859
C06610=1177.637,75.903,-49.918,-179.206,6.085,148.858
C06611=1177.632,76.152,-49.934,-179.203,6.086,148.858
C06612=1177.627,76.401,-49.952,-179.200,6.087,148.857
C06613=1177.622,76.650,-49.969,-179.198,6.088,148.857
C06614=1177.617,76.900,-49.986,-179.195,6.090,148.856
C06615=1177.612,77.149,-50.004,-179.193,6.091,148.855
C06616=1177.608,77.399,-50.021,-179.190,6.092,148.855
C06617=1177.603,77.648,-50.038,-179.187,6.093,148.854
C06618=1177.598,77.897,-50.055,-179.185,6.093,148.854
C06619=1177.593,78.146,-50.072,-179.182,6.095,148.853
C06620=1177.587,78.396,-50.089,-179.179,6.096,148.853
C06621=1177.583,78.645,-50.107,-179.177,6.097,148.852
C06622=1177.578,78.895,-50.124,-179.174,6.098,148.852
C06623=1177.573,79.144,-50.142,-179.171,6.100,148.851
C06624=1177.569,79.394,-50.159,-179.169,6.100,148.850
C06625=1177.563,79.643,-50.176,-179.166,6.102,148.850
C06626=1177.558,79.892,-50.194,-179.164,6.103,148.850
C06627=1177.553,80.160,-50.212,-179.161,6.104,148.849
C06628=1177.548,80.429,-50.230,-179.158,6.105,148.848
C06629=1177.542,80.697,-50.249,-179.155,6.106,148.848
C06630=1177.537,80.966,-50.268,-179.152,6.108,148.847
C06631=1177.533,81.214,-50.285,-179.149,6.108,148.847
C06632=1177.527,81.464,-50.303,-179.147,6.110,148.846
C06633=1177.522,81.713,-50.321,-179.145,6.111,148.846
C06634=1177.517,81.963,-50.338,-179.141,6.112,148.845
C06635=1177.513,82.212,-50.355,-179.139,6.113,148.845
C06636=1177.508,82.462,-50.373,-179.137,6.113,148.844
C06637=1177.503,82.711,-50.391,-179.134,6.115,148.844
C06638=1177.498,82.961,-50.407,-179.131,6.116,148.843
C06639=1177.494,83.210,-50.425,-179.129,6.117,148.843
C06640=1177.488,83.460,-50.442,-179.126,6.118,148.842
C06641=1177.483,83.708,-50.460,-179.123,6.120,148.841
C06642=1177.478,83.958,-50.477,-179.121,6.120,148.841
C06643=1177.473,84.207,-50.495,-179.118,6.122,148.840
C06644=1177.468,84.456,-50.513,-179.116,6.123,148.840
C06645=1177.463,84.706,-50.530,-179.112,6.124,148.839
C06646=1177.458,84.955,-50.548,-179.110,6.125,148.839
C06647=1177.453,85.204,-50.566,-179.107,6.126,148.838
C06648=1177.449,85.453,-50.583,-179.105,6.127,148.838
C06649=1177.444,85.703,-50.601,-179.102,6.129,148.837
C06650=1177.439,85.952,-50.618,-179.100,6.130,148.837
C06651=1177.434,86.202,-50.636,-179.096,6.131,148.836
C06652=1177.429,86.451,-50.654,-179.094,6.132,148.836
C06653=1177.425,86.700,-50.671,-179.092,6.134,148.835
C06654=1177.420,86.949,-50.688,-179.089,6.134,148.835
C06655=1177.415,87.199,-50.706,-179.086,6.136,148.834
C06656=1177.410,87.448,-50.724,-179.084,6.136,148.834
C06657=1177.405,87.698,-50.742,-179.081,6.138,148.833
C06658=1177.400,87.947,-50.760,-179.078,6.139,148.832
C06659=1177.395,88.196,-50.778,-179.076,6.140,148.832
C06660=1177.390,88.445,-50.796,-179.073,6.141,148.832
C06661=1177.385,88.696,-50.813,-179.070,6.143,148.831
C06662=1177.381,88.945,-50.831,-179.068,6.143,148.831
C06663=1177.376,89.194,-50.849,-179.065,6.145,148.830
C06664=1177.371,89.443,-50.867,-179.063,6.146,148.829
C06665=1177.366,89.692,-50.885,-179.059,6.147,148.829
C06666=1177.361,89.942,-50.902,-179.057,6.148,148.828
C06667=1177.356,90.191,-50.920,-179.055,6.150,148.828
C06668=1177.351,90.440,-50.938,-179.052,6.150,148.827
C06669=1177.346,90.689,-50.956,-179.049,6.152,148.827
C06670=1177.341,90.939,-50.974,-179.047,6.152,148.826
C06671=1177.337,91.188,-50.992,-179.044,6.154,148.826
C06672=1177.331,91.438,-51.009,-179.041,6.156,148.825
C06673=1177.326,91.687,-51.027,-179.039,6.156,148.825
C06674=1177.321,91.936,-51.045,-179.036,6.158,148.824
C06675=1177.317,92.186,-51.063,-179.033,6.159,148.824
C06676=1177.312,92.435,-51.081,-179.031,6.160,148.823
C06677=1177.307,92.684,-51.099,-179.028,6.161,148.823
C06678=1177.302,92.933,-51.117,-179.025,6.163,148.822
C06679=1177.298,93.182,-51.135,-179.023,6.164,148.822
C06680=1177.293,93.432,-51.153,-179.020,6.165,148.821
C06681=1177.288,93.681,-51.171,-179.018,6.166,148.821
C06682=1177.283,93.930,-51.189,-179.015,6.167,148.820
C06683=1177.278,94.180,-51.208,-179.012,6.168,148.820
C06684=1177.274,94.429,-51.226,-179.010,6.170,148.819
C06685=1177.269,94.678,-51.243,-179.006,6.171,148.819
C06686=1177.264,94.927,-51.261,-179.004,6.172,148.818
C06687=1177.259,95.177,-51.279,-179.001,6.173,148.818
C06688=1177.254,95.426,-51.297,-178.999,6.174,148.817
C06689=1177.249,95.676,-51.316,-178.996,6.176,148.817
C06690=1177.244,95.925,-51.334,-178.994,6.177,148.816
C06691=1177.239,96.174,-51.352,-178.991,6.178,148.816
C06692=1177.234,96.423,-51.370,-178.988,6.179,148.815
C06693=1177.229,96.673,-51.388,-178.986,6.181,148.815
C06694=1177.224,96.922,-51.406,-178.983,6.182,148.814
C06695=1177.220,97.172,-51.425,-178.980,6.183,148.814
C06696=1177.215,97.421,-51.443,-178.978,6.185,148.813
C06697=1177.210,97.670,-51.462,-178.975,6.185,148.813
C06698=1177.205,97.919,-51.480,-178.972,6.187,148.812
C06699=1177.200,98.168,-51.498,-178.970,6.188,148.812
C06700=1177.196,98.418,-51.516,-178.967,6.189,148.811
C06701=1177.191,98.667,-51.534,-178.964,6.191,148.811
C06702=1177.186,98.916,-51.552,-178.962,6.192,148.810
C06703=1177.180,99.166,-51.571,-178.959,6.193,148.810
C06704=1177.176,99.415,-51.590,-178.957,6.194,148.809
C06705=1177.171,99.664,-51.608,-178.954,6.196,148.809
C06706=1177.166,99.913,-51.626,-178.951,6.197,148.808
C06707=1177.161,100.163,-51.644,-178.949,6.198,148.808
C06708=1177.156,100.411,-51.663,-178.945,6.199,148.807
C06709=1177.152,100.661,-51.681,-178.943,6.200,148.807
C06710=1177.147,100.910,-51.699,-178.941,6.202,148.806
C06711=1177.142,101.160,-51.717,-178.938,6.203,148.806
C06712=1177.137,101.409,-51.737,-178.935,6.204,148.805
C06713=1177.132,101.658,-51.755,-178.933,6.206,148.805
C06714=1177.127,101.908,-51.773,-178.930,6.207,148.804
C06715=1177.122,102.157,-51.791,-178.927,6.208,148.804
C06716=1177.118,102.406,-51.811,-178.925,6.209,148.803
C06717=1177.113,102.656,-51.829,-178.922,6.211,148.803
C06718=1177.108,102.905,-51.847,-178.919,6.212,148.802
C06719=1177.104,103.154,-51.866,-178.917,6.213,148.802
C06720=1177.098,103.403,-51.884,-178.914,6.215,148.801
C06721=1177.093,103.653,-51.902,-178.911,6.216,148.801
C06722=1177.089,103.901,-51.921,-178.909,6.217,148.800
C06723=1177.084,104.151,-51.940,-178.906,6.219,148.800
C06724=1177.079,104.400,-51.958,-178.904,6.219,148.799
C06725=1177.074,104.649,-51.976,-178.900,6.221,148.799
C06726=1177.069,104.899,-51.995,-178.898,6.223,148.798
C06727=1177.064,105.148,-52.014,-178.896,6.223,148.798
C06728=1177.060,105.397,-52.032,-178.892,6.225,148.797
C06729=1177.055,105.647,-52.052,-178.890,6.226,148.797
C06730=1177.050,105.896,-52.070,-178.888,6.227,148.796
C06731=1177.044,106.164,-52.090,-178.884,6.229,148.796
C06732=1177.040,106.433,-52.110,-178.882,6.231,148.795
C06733=1177.034,106.701,-52.130,-178.878,6.232,148.795
C06734=1177.029,106.969,-52.151,-178.876,6.233,148.794
C06735=1177.024,107.219,-52.169,-178.873,6.234,148.794
C06736=1177.020,107.468,-52.188,-178.870,6.236,148.793
C06737=1177.014,107.717,-52.207,-178.868,6.237,148.793
C06738=1177.010,107.966,-52.226,-178.865,6.238,148.792
C06739=1177.004,108.216,-52.244,-178.862,6.240,148.792
C06740=1177.000,108.465,-52.263,-178.860,6.241,148.791
C06741=1176.995,108.715,-52.282,-178.857,6.242,148.791
C06742=1176.990,108.963,-52.301,-178.854,6.244,148.790
C06743=1176.986,109.212,-52.320,-178.852,6.245,148.790
C06744=1176.980,109.462,-52.338,-178.849,6.246,148.789
C06745=1176.976,109.711,-52.357,-178.847,6.247,148.789
C06746=1176.971,109.961,-52.376,-178.844,6.249,148.788
C06747=1176.966,110.209,-52.394,-178.841,6.250,148.788
C06748=1176.961,110.459,-52.414,-178.839,6.251,148.787
C06749=1176.957,110.708,-52.432,-178.836,6.253,148.787
C06750=1176.952,110.957,-52.452,-178.833,6.254,148.786
C06751=1176.947,111.206,-52.470,-178.831,6.255,148.786
C06752=1176.942,111.456,-52.489,-178.828,6.257,148.786
C06753=1176.938,111.705,-52.508,-178.825,6.258,148.785
C06754=1176.933,111.954,-52.528,-178.823,6.259,148.785
C06755=1176.927,112.204,-52.546,-178.820,6.261,148.784
C06756=1176.923,112.452,-52.565,-178.817,6.262,148.784
C06757=1176.918,112.702,-52.585,-178.815,6.263,148.783
C06758=1176.913,112.950,-52.603,-178.812,6.265,148.783
C06759=1176.908,113.201,-52.622,-178.809,6.267,148.782
C06760=1176.904,113.449,-52.641,-178.807,6.267,148.782
C06761=1176.899,113.699,-52.661,-178.804,6.269,148.781
C06762=1176.893,113.948,-52.680,-178.801,6.271,148.781
C06763=1176.889,114.198,-52.698,-178.799,6.271,148.780
C06764=1176.884,114.446,-52.718,-178.796,6.273,148.780
C06765=1176.879,114.696,-52.737,-178.793,6.275,148.779
C06766=1176.874,114.945,-52.756,-178.791,6.276,148.779
C06767=1176.870,115.194,-52.776,-178.788,6.277,148.778
C06768=1176.865,115.443,-52.794,-178.785,6.279,148.778
C06769=1176.860,115.693,-52.813,-178.783,6.280,148.778
C06770=1176.855,115.942,-52.833,-178.780,6.281,148.777
C06771=1176.851,116.191,-52.852,-178.777,6.283,148.777
C06772=1176.845,116.440,-52.871,-178.775,6.284,148.776
C06773=1176.841,116.689,-52.891,-178.772,6.285,148.776
C06774=1176.837,116.939,-52.910,-178.769,6.287,148.775
C06775=1176.831,117.188,-52.929,-178.767,6.288,148.775
C06776=1176.827,117.437,-52.949,-178.764,6.289,148.774
C06777=1176.821,117.687,-52.967,-178.761,6.291,148.774
C06778=1176.817,117.936,-52.986,-178.758,6.293,148.773
C06779=1176.812,118.185,-53.005,-178.756,6.294,148.773
C06780=1176.807,118.434,-53.025,-178.754,6.295,148.772
C06781=1176.803,118.684,-53.044,-178.750,6.297,148.772
C06782=1176.797,118.932,-53.063,-178.748,6.298,148.771
C06783=1176.793,119.182,-53.083,-178.746,6.299,148.771
C06784=1176.787,119.431,-53.102,-178.742,6.301,148.770
C06785=1176.783,119.680,-53.121,-178.740,6.302,148.770
C06786=1176.778,119.929,-53.141,-178.737,6.304,148.770
C06787=1176.773,120.179,-53.160,-178.735,6.305,148.769
C06788=1176.768,120.428,-53.180,-178.732,6.306,148.769
C06789=1176.763,120.677,-53.199,-178.729,6.308,148.768
C06790=1176.759,120.926,-53.219,-178.727,6.309,148.768
C06791=1176.755,121.175,-53.239,-178.724,6.311,148.767
C06792=1176.749,121.424,-53.258,-178.721,6.312,148.767
C06793=1176.745,121.674,-53.278,-178.718,6.314,148.766
C06794=1176.739,121.922,-53.297,-178.716,6.315,148.766
C06795=1176.735,122.172,-53.316,-178.713,6.316,148.766
C06796=1176.731,122.421,-53.336,-178.710,6.318,148.765
C06797=1176.725,122.670,-53.355,-178.708,6.320,148.764
C06798=1176.720,122.920,-53.375,-178.705,6.321,148.764
C06799=1176.716,123.169,-53.395,-178.703,6.322,148.764
C06800=1176.711,123.418,-53.414,-178.700,6.324,148.763
C06801=1176.706,123.667,-53.434,-178.697,6.325,148.763
C06802=1176.702,123.916,-53.453,-178.695,6.326,148.762
C06803=1176.697,124.165,-53.472,-178.692,6.328,148.762
C06804=1176.692,124.414,-53.493,-178.689,6.329,148.761
C06805=1176.687,124.664,-53.512,-178.686,6.331,148.761
C06806=1176.682,124.913,-53.532,-178.684,6.332,148.760
C06807=1176.677,125.162,-53.551,-178.681,6.334,148.760
C06808=1176.673,125.411,-53.572,-178.679,6.336,148.760
C06809=1176.668,125.661,-53.591,-178.675,6.337,148.759
C06810=1176.663,125.910,-53.611,-178.673,6.338,148.759
C06811=1176.658,126.159,-53.630,-178.671,6.340,148.758
C06812=1176.654,126.408,-53.651,-178.668,6.341,148.758
C06813=1176.648,126.657,-53.670,-178.665,6.343,148.757
C06814=1176.644,126.907,-53.690,-178.663,6.344,148.757
C06815=1176.640,127.155,-53.709,-178.660,6.345,148.756
C06816=1176.635,127.405,-53.729,-178.657,6.347,148.756
C06817=1176.630,127.654,-53.748,-178.654,6.349,148.756
C06818=1176.625,127.903,-53.769,-178.651,6.350,148.755
C06819=1176.621,128.152,-53.788,-178.649,6.351,148.755
C06820=1176.616,128.402,-53.808,-178.646,6.353,148.754
C06821=1176.611,128.650,-53.828,-178.644,6.355,148.754
C06822=1176.606,128.900,-53.848,-178.641,6.356,148.753
C06823=1176.602,129.148,-53.868,-178.638,6.357,148.753
C06824=1176.596,129.398,-53.888,-178.636,6.359,148.752
C06825=1176.591,129.648,-53.908,-178.633,6.360,148.752
C06826=1176.586,129.896,-53.928,-178.630,6.362,148.752
C06827=1176.582,130.146,-53.948,-178.627,6.364,148.751
C06828=1176.577,130.395,-53.968,-178.625,6.365,148.751
C06829=1176.572,130.644,-53.988,-178.622,6.366,148.750
C06830=1176.568,130.893,-54.008,-178.620,6.368,148.750
C06831=1176.563,131.142,-54.027,-178.617,6.370,148.749
C06832=1176.558,131.391,-54.048,-178.614,6.371,148.749
C06833=1176.553,131.641,-54.067,-178.612,6.372,148.748
C06834=1176.549,131.890,-54.088,-178.609,6.374,148.748
C06835=1176.543,132.159,-54.109,-178.606,6.376,148.748
C06836=1176.538,132.427,-54.131,-178.603,6.377,148.747
C06837=1176.533,132.695,-54.153,-178.600,6.379,148.747
C06838=1176.528,132.964,-54.174,-178.598,6.380,148.746
C06839=1176.524,133.213,-54.194,-178.594,6.382,148.746
C06840=1176.518,133.463,-54.215,-178.592,6.384,148.745
C06841=1176.513,133.711,-54.235,-178.589,6.385,148.745
C06842=1176.509,133.960,-54.255,-178.587,6.386,148.744
C06843=1176.504,134.210,-54.275,-178.584,6.388,148.744
C06844=1176.500,134.459,-54.295,-178.582,6.390,148.744
C06845=1176.495,134.708,-54.315,-178.578,6.391,148.743
C06846=1176.490,134.958,-54.336,-178.576,6.393,148.743
C06847=1176.485,135.206,-54.356,-178.573,6.395,148.742
C06848=1176.480,135.455,-54.376,-178.571,6.396,148.742
C06849=1176.475,135.704,-54.396,-178.568,6.397,148.741
C06850=1176.470,135.954,-54.417,-178.565,6.399,148.741
C06851=1176.466,136.202,-54.437,-178.562,6.400,148.740
C06852=1176.461,136.452,-54.457,-178.560,6.402,148.740
C06853=1176.457,136.701,-54.477,-178.557,6.404,148.740
C06854=1176.451,136.950,-54.498,-178.555,6.405,148.739
C06855=1176.447,137.199,-54.518,-178.552,6.407,148.739
C06856=1176.442,137.449,-54.538,-178.549,6.408,148.738
C06857=1176.438,137.698,-54.558,-178.546,6.410,148.738
C06858=1176.433,137.947,-54.579,-178.543,6.411,148.737
C06859=1176.428,138.196,-54.600,-178.541,6.413,148.737
C06860=1176.423,138.445,-54.619,-178.539,6.414,148.737
C06861=1176.418,138.694,-54.640,-178.536,6.416,148.736
C06862=1176.413,138.943,-54.660,-178.533,6.418,148.736
C06863=1176.409,139.192,-54.681,-178.530,6.419,148.735
C06864=1176.404,139.441,-54.702,-178.527,6.421,148.735
C06865=1176.399,139.690,-54.722,-178.525,6.423,148.735
C06866=1176.395,139.939,-54.742,-178.522,6.424,148.734
C06867=1176.389,140.189,-54.763,-178.520,6.425,148.734
C06868=1176.385,140.438,-54.783,-178.517,6.427,148.733
C06869=1176.380,140.687,-54.803,-178.514,6.429,148.733
C06870=1176.375,140.936,-54.824,-178.511,6.430,148.732
C06871=1176.371,141.185,-54.845,-178.509,6.432,148.732
C06872=1176.366,141.434,-54.865,-178.506,6.434,148.732
C06873=1176.361,141.683,-54.886,-178.503,6.435,148.731
C06874=1176.357,141.932,-54.907,-178.501,6.436,148.731
C06875=1176.352,142.182,-54.927,-178.498,6.438,148.730
C06876=1176.347,142.430,-54.948,-178.496,6.440,148.730
C06877=1176.343,142.679,-54.968,-178.493,6.442,148.730
C06878=1176.338,142.929,-54.989,-178.490,6.443,148.729
C06879=1176.333,143.178,-55.010,-178.487,6.445,148.729
C06880=1176.328,143.427,-55.031,-178.484,6.446,148.728
C06881=1176.324,143.676,-55.051,-178.482,6.448,148.728
C06882=1176.318,143.925,-55.072,-178.480,6.449,148.727
C06883=1176.314,144.174,-55.092,-178.477,6.451,148.727
C06884=1176.309,144.424,-55.114,-178.474,6.453,148.727
C06885=1176.305,144.673,-55.134,-178.472,6.454,148.726
C06886=1176.300,144.922,-55.154,-178.469,6.456,148.726
C06887=1176.295,145.171,-55.175,-178.466,6.458,148.725
C06888=1176.291,145.420,-55.196,-178.463,6.459,148.725
C06889=1176.286,145.669,-55.217,-178.460,6.461,148.725
C06890=1176.282,145.918,-55.238,-178.458,6.463,148.724
C06891=1176.276,146.167,-55.259,-178.455,6.465,148.724
C06892=1176.271,146.416,-55.280,-178.453,6.465,148.723
C06893=1176.267,146.665,-55.300,-178.450,6.467,148.723
C06894=1176.262,146.914,-55.321,-178.447,6.469,148.723
C06895=1176.257,147.163,-55.341,-178.445,6.471,148.722
C06896=1176.253,147.413,-55.363,-178.442,6.472,148.722
C06897=1176.248,147.662,-55.384,-178.439,6.474,148.721
C06898=1176.243,147.911,-55.405,-178.436,6.476,148.721
C06899=1176.239,148.160,-55.425,-178.433,6.477,148.721
C06900=1176.234,148.409,-55.446,-178.431,6.479,148.720
C06901=1176.229,148.658,-55.468,-178.428,6.481,148.720
C06902=1176.224,148.907,-55.488,-178.425,6.483,148.719
C06903=1176.219,149.156,-55.509,-178.423,6.484,148.719
C06904=1176.215,149.405,-55.531,-178.421,6.485,148.719
C06905=1176.210,149.654,-55.552,-178.418,6.487,148.718
C06906=1176.205,149.904,-55.572,-178.415,6.489,148.718
C06907=1176.201,150.152,-55.593,-178.412,6.491,148.717
C06908=1176.196,150.401,-55.615,-178.410,6.492,148.717
C06909=1176.191,150.650,-55.636,-178.407,6.494,148.716
C06910=1176.187,150.900,-55.656,-178.404,6.496,148.716
C06911=1176.182,151.149,-55.678,-178.401,6.497,148.716
C06912=1176.177,151.398,-55.699,-178.399,6.499,148.715
C06913=1176.173,151.646,-55.720,-178.396,6.501,148.715
C06914=1176.168,151.896,-55.741,-178.393,6.503,148.715
C06915=1176.162,152.145,-55.762,-178.390,6.504,148.714
C06916=1176.158,152.394,-55.784,-178.388,6.506,148.714
C06917=1176.154,152.643,-55.804,-178.385,6.508,148.713
C06918=1176.149,152.892,-55.826,-178.383,6.509,148.713
C06919=1176.144,153.141,-55.847,-178.380,6.511,148.713
C06920=1176.139,153.391,-55.868,-178.378,6.512,148.712
C06921=1176.135,153.639,-55.889,-178.375,6.514,148.712
C06922=1176.130,153.889,-55.910,-178.372,6.516,148.712
C06923=1176.125,154.137,-55.932,-178.370,6.518,148.711
C06924=1176.120,154.386,-55.953,-178.367,6.519,148.711
C06925=1176.116,154.635,-55.974,-178.364,6.521,148.710
C06926=1176.111,154.885,-55.995,-178.361,6.523,148.710
C06927=1176.106,155.133,-56.017,-178.358,6.524,148.709
C06928=1176.101,155.383,-56.038,-178.356,6.526,148.709
C06929=1176.097,155.632,-56.060,-178.353,6.528,148.709
C06930=1176.093,155.880,-56.081,-178.350,6.529,148.708
C06931=1176.087,156.130,-56.102,-178.348,6.531,148.708
C06932=1176.083,156.379,-56.124,-178.345,6.533,148.708
C06933=1176.078,156.628,-56.145,-178.342,6.535,148.707
C06934=1176.073,156.877,-56.167,-178.339,6.537,148.707
C06935=1176.068,157.125,-56.189,-178.337,6.538,148.706
C06936=1176.064,157.375,-56.209,-178.334,6.540,148.706
C06937=1176.060,157.624,-56.231,-178.331,6.542,148.706
C06938=1176.054,157.873,-56.252,-178.329,6.544,148.705
C06939=1176.049,158.142,-56.276,-178.326,6.545,148.705
C06940=1176.044,158.411,-56.299,-178.323,6.547,148.705
C06941=1176.039,158.680,-56.322,-178.321,6.549,148.704
C06942=1176.035,158.949,-56.346,-178.317,6.551,148.704
C06943=1176.029,159.198,-56.367,-178.314,6.553,148.703
C06944=1176.025,159.447,-56.389,-178.312,6.555,148.703
C06945=1176.020,159.696,-56.410,-178.309,6.556,148.703
C06946=1176.015,159.945,-56.431,-178.306,6.558,148.702
C06947=1176.011,160.194,-56.453,-178.303,6.560,148.702
C06948=1176.006,160.443,-56.475,-178.301,6.562,148.701
C06949=1176.001,160.692,-56.497,-178.298,6.563,148.701
C06950=1175.997,160.941,-56.519,-178.295,6.565,148.701
C06951=1175.992,161.190,-56.540,-178.293,6.567,148.700
C06952=1175.987,161.440,-56.562,-178.290,6.569,148.700
C06953=1175.982,161.688,-56.583,-178.287,6.570,148.700
C06954=1175.978,161.937,-56.605,-178.285,6.572,148.699
C06955=1175.973,162.186,-56.627,-178.282,6.574,148.699
C06956=1175.968,162.435,-56.648,-178.279,6.576,148.698
C06957=1175.963,162.684,-56.670,-178.277,6.578,148.698
C06958=1175.959,162.933,-56.692,-178.274,6.579,148.698
C06959=1175.954,163.182,-56.714,-178.271,6.581,148.697
C06960=1175.950,163.431,-56.736,-178.269,6.583,148.697
C06961=1175.945,163.680,-56.757,-178.266,6.585,148.697
C06962=1175.941,163.929,-56.779,-178.263,6.586,148.696
C06963=1175.936,164.178,-56.801,-178.261,6.588,148.696
C06964=1175.931,164.427,-56.823,-178.258,6.590,148.696
C06965=1175.927,164.676,-56.845,-178.256,6.592,148.695
C06966=1175.922,164.925,-56.866,-178.253,6.594,148.695
C06967=1175.918,165.174,-56.889,-178.250,6.595,148.695
C06968=1175.913,165.423,-56.910,-178.248,6.597,148.694
C06969=1175.908,165.672,-56.932,-178.245,6.599,148.694
C06970=1175.904,165.921,-56.954,-178.242,6.601,148.693
C06971=1175.899,166.170,-56.977,-178.239,6.603,148.693
C06972=1175.894,166.419,-56.998,-178.237,6.604,148.693
C06973=1175.889,166.668,-57.020,-178.234,6.606,148.692
C06974=1175.885,166.917,-57.042,-178.231,6.608,148.692
C06975=1175.880,167.166,-57.064,-178.229,6.610,148.692
C06976=1175.875,167.415,-57.086,-178.226,6.611,148.691
C06977=1175.871,167.664,-57.108,-178.223,6.613,148.691
C06978=1175.866,167.913,-57.130,-178.221,6.615,148.690
C06979=1175.861,168.163,-57.152,-178.218,6.617,148.690
C06980=1175.856,168.411,-57.174,-178.215,6.619,148.690
C06981=1175.852,168.661,-57.196,-178.212,6.621,148.689
C06982=1175.848,168.909,-57.218,-178.209,6.623,148.689
C06983=1175.843,169.158,-57.241,-178.207,6.625,148.689
C06984=1175.838,169.407,-57.263,-178.204,6.626,148.688
C06985=1175.833,169.656,-57.285,-178.201,6.628,148.688
C06986=1175.829,169.905,-57.306,-178.199,6.630,148.688
C06987=1175.824,170.154,-57.329,-178.196,6.632,148.687
C06988=1175.819,170.402,-57.351,-178.194,6.634,148.687
C06989=1175.815,170.652,-57.373,-178.191,6.636,148.687
C06990=1175.810,170.900,-57.395,-178.188,6.637,148.686
C06991=1175.805,171.150,-57.418,-178.186,6.639,148.686
C06992=1175.800,171.398,-57.440,-178.183,6.641,148.686
C06993=1175.796,171.647,-57.462,-178.180,6.643,148.685
C06994=1175.791,171.897,-57.485,-178.178,6.644,148.685
C06995=1175.786,172.146,-57.506,-178.174,6.647,148.685
C06996=1175.782,172.395,-57.529,-178.172,6.649,148.684
C06997=1175.777,172.643,-57.551,-178.169,6.650,148.684
C06998=1175.772,172.893,-57.574,-178.166,6.652,148.683
C06999=1175.768,173.142,-57.596,-178.164,6.654,148.683
C07000=1175.764,173.390,-57.618,-178.161,6.656,148.683
C07001=1175.759,173.640,-57.641,-178.159,6.658,148.683
C07002=1175.754,173.888,-57.663,-178.156,6.660,148.682
C07003=1175.749,174.137,-57.686,-178.153,6.661,148.682
C07004=1175.745,174.386,-57.708,-178.151,6.663,148.681
C07005=1175.740,174.635,-57.730,-178.148,6.665,148.681
C07006=1175.735,174.885,-57.753,-178.145,6.668,148.681
C07007=1175.731,175.133,-57.775,-178.142,6.669,148.680
C07008=1175.726,175.382,-57.797,-178.139,6.671,148.680
C07009=1175.722,175.631,-57.821,-178.137,6.673,148.680
C07010=1175.717,175.880,-57.842,-178.135,6.675,148.680
C07011=1175.712,176.129,-57.866,-178.132,6.677,148.679
C07012=1175.708,176.378,-57.888,-178.129,6.679,148.679
C07013=1175.702,176.626,-57.911,-178.127,6.680,148.678
C07014=1175.698,176.876,-57.933,-178.124,6.682,148.678
C07015=1175.694,177.124,-57.955,-178.121,6.685,148.678
C07016=1175.689,177.373,-57.978,-178.118,6.686,148.677
C07017=1175.685,177.622,-58.001,-178.115,6.688,148.677
C07018=1175.680,177.872,-58.023,-178.113,6.690,148.677
C07019=1175.676,178.120,-58.046,-178.110,6.692,148.677
C07020=1175.670,178.369,-58.068,-178.108,6.694,148.676
C07021=1175.666,178.618,-58.091,-178.105,6.696,148.676
C07022=1175.661,178.868,-58.114,-178.102,6.697,148.675
C07023=1175.657,179.116,-58.136,-178.099,6.700,148.675
C07024=1175.652,179.365,-58.159,-178.096,6.702,148.675
C07025=1175.648,179.614,-58.181,-178.094,6.704,148.674
C07026=1175.643,179.863,-58.205,-178.092,6.706,148.674
C07027=1175.638,180.111,-58.228,-178.089,6.707,148.674
C07028=1175.633,180.361,-58.250,-178.086,6.709,148.673
C07029=1175.629,180.610,-58.273,-178.083,6.711,148.673
C07030=1175.625,180.859,-58.296,-178.080,6.714,148.673
C07031=1175.619,181.107,-58.318,-178.078,6.715,148.672
C07032=1175.615,181.356,-58.341,-178.075,6.717,148.672
C07033=1175.610,181.605,-58.364,-178.073,6.719,148.672
C07034=1175.606,181.854,-58.388,-178.070,6.721,148.672
C07035=1175.601,182.103,-58.409,-178.067,6.723,148.671
C07036=1175.596,182.352,-58.433,-178.065,6.725,148.671
C07037=1175.592,182.601,-58.455,-178.061,6.727,148.671
C07038=1175.587,182.850,-58.479,-178.059,6.729,148.670
C07039=1175.582,183.099,-58.501,-178.056,6.731,148.670
C07040=1175.578,183.347,-58.524,-178.054,6.733,148.670
C07041=1175.573,183.596,-58.547,-178.051,6.735,148.669
C07042=1175.568,183.845,-58.571,-178.048,6.736,148.669
C07043=1175.564,184.115,-58.595,-178.045,6.739,148.669
C07044=1175.559,184.385,-58.620,-178.043,6.741,148.668
C07045=1175.554,184.654,-58.645,-178.039,6.743,148.668
C07046=1175.549,184.924,-58.670,-178.037,6.745,148.668
C07047=1175.544,185.173,-58.693,-178.034,6.747,148.667
C07048=1175.539,185.422,-58.716,-178.031,6.749,148.667
C07049=1175.535,185.671,-58.739,-178.029,6.752,148.667
C07050=1175.530,185.919,-58.762,-178.026,6.753,148.666
C07051=1175.525,186.168,-58.785,-178.023,6.755,148.666
C07052=1175.521,186.417,-58.808,-178.020,6.757,148.666
C07053=1175.517,186.666,-58.832,-178.018,6.759,148.665
C07054=1175.512,186.915,-58.855,-178.015,6.761,148.665
C07055=1175.507,187.164,-58.878,-178.012,6.763,148.665
C07056=1175.503,187.413,-58.901,-178.010,6.765,148.665
C07057=1175.498,187.661,-58.924,-178.007,6.767,148.664
C07058=1175.493,187.910,-58.947,-178.004,6.769,148.664
C07059=1175.489,188.159,-58.971,-178.001,6.771,148.663
C07060=1175.484,188.408,-58.994,-177.999,6.773,148.663
C07061=1175.480,188.657,-59.017,-177.996,6.775,148.663
C07062=1175.475,188.906,-59.040,-177.994,6.777,148.663
C07063=1175.471,189.155,-59.064,-177.991,6.779,148.662
C07064=1175.466,189.404,-59.087,-177.988,6.781,148.662
C07065=1175.461,189.653,-59.110,-177.985,6.784,148.662
C07066=1175.456,189.902,-59.134,-177.983,6.785,148.661
C07067=1175.451,190.150,-59.157,-177.980,6.787,148.661
C07068=1175.447,190.399,-59.179,-177.977,6.789,148.661
C07069=1175.442,190.648,-59.203,-177.975,6.792,148.661
C07070=1175.438,190.896,-59.227,-177.972,6.794,148.660
C07071=1175.433,191.145,-59.250,-177.969,6.795,148.660
C07072=1175.429,191.394,-59.274,-177.967,6.797,148.660
C07073=1175.424,191.643,-59.297,-177.964,6.799,148.659
C07074=1175.419,191.892,-59.320,-177.961,6.802,148.659
C07075=1175.415,192.141,-59.344,-177.959,6.804,148.659
C07076=1175.410,192.390,-59.368,-177.956,6.805,148.658
C07077=1175.405,192.639,-59.391,-177.953,6.807,148.658
C07078=1175.401,192.888,-59.414,-177.950,6.810,148.658
C07079=1175.396,193.137,-59.438,-177.948,6.812,148.658
C07080=1175.392,193.385,-59.461,-177.945,6.814,148.657
C07081=1175.388,193.634,-59.485,-177.942,6.816,148.657
C07082=1175.383,193.883,-59.508,-177.940,6.818,148.657
C07083=1175.379,194.132,-59.532,-177.937,6.820,148.656
C07084=1175.374,194.381,-59.555,-177.934,6.822,148.656
C07085=1175.369,194.630,-59.579,-177.932,6.824,148.656
C07086=1175.365,194.878,-59.603,-177.929,6.826,148.656
C07087=1175.360,195.127,-59.626,-177.926,6.829,148.655
C07088=1175.355,195.376,-59.650,-177.923,6.830,148.655
C07089=1175.351,195.625,-59.674,-177.921,6.832,148.655
C07090=1175.346,195.874,-59.698,-177.919,6.834,148.654
C07091=1175.341,196.123,-59.721,-177.915,6.837,148.654
C07092=1175.337,196.371,-59.745,-177.913,6.839,148.654
C07093=1175.332,196.620,-59.768,-177.910,6.840,148.653
C07094=1175.327,196.869,-59.792,-177.908,6.843,148.653
C07095=1175.323,197.118,-59.816,-177.905,6.845,148.653
C07096=1175.318,197.366,-59.840,-177.902,6.847,148.653
C07097=1175.314,197.616,-59.864,-177.899,6.849,148.652
C07098=1175.310,197.864,-59.888,-177.897,6.852,148.652
C07099=1175.305,198.113,-59.911,-177.894,6.853,148.652
C07100=1175.300,198.362,-59.934,-177.891,6.855,148.651
C07101=1175.296,198.611,-59.958,-177.888,6.857,148.651
C07102=1175.291,198.860,-59.983,-177.886,6.860,148.651
C07103=1175.286,199.109,-60.006,-177.883,6.862,148.651
C07104=1175.282,199.357,-60.031,-177.880,6.864,148.650
C07105=1175.277,199.606,-60.054,-177.878,6.866,148.650
C07106=1175.273,199.854,-60.078,-177.875,6.868,148.650
C07107=1175.269,200.104,-60.102,-177.872,6.870,148.650
C07108=1175.264,200.353,-60.126,-177.870,6.872,148.649
C07109=1175.259,200.601,-60.150,-177.867,6.875,148.649
C07110=1175.254,200.850,-60.174,-177.864,6.877,148.649
C07111=1175.250,201.099,-60.198,-177.862,6.878,148.648
C07112=1175.245,201.348,-60.221,-177.859,6.880,148.648
C07113=1175.241,201.596,-60.245,-177.856,6.883,148.648
C07114=1175.236,201.846,-60.270,-177.853,6.885,148.648
C07115=1175.232,202.095,-60.294,-177.851,6.887,148.647
C07116=1175.227,202.343,-60.318,-177.848,6.890,148.647
C07117=1175.223,202.592,-60.342,-177.845,6.891,148.647
C07118=1175.218,202.840,-60.367,-177.843,6.893,148.647
C07119=1175.213,203.089,-60.390,-177.840,6.895,148.646
C07120=1175.209,203.338,-60.414,-177.837,6.898,148.646
C07121=1175.205,203.587,-60.438,-177.835,6.900,148.646
C07122=1175.199,203.836,-60.462,-177.832,6.902,148.646
C07123=1175.195,204.085,-60.486,-177.829,6.904,148.645
C07124=1175.191,204.333,-60.511,-177.826,6.906,148.645
C07125=1175.186,204.582,-60.536,-177.824,6.908,148.645
C07126=1175.182,204.831,-60.560,-177.821,6.911,148.644
C07127=1175.177,205.080,-60.583,-177.818,6.913,148.644
C07128=1175.172,205.329,-60.608,-177.816,6.915,148.644
C07129=1175.168,205.578,-60.632,-177.813,6.917,148.644
C07130=1175.164,205.826,-60.656,-177.810,6.919,148.643
C07131=1175.159,206.075,-60.681,-177.808,6.921,148.643
C07132=1175.154,206.323,-60.705,-177.805,6.924,148.643
C07133=1175.150,206.572,-60.729,-177.802,6.926,148.643
C07134=1175.145,206.822,-60.753,-177.800,6.928,148.642
C07135=1175.141,207.070,-60.777,-177.797,6.930,148.642
C07136=1175.135,207.319,-60.802,-177.794,6.932,148.642
C07137=1175.132,207.568,-60.826,-177.792,6.934,148.642
C07138=1175.127,207.816,-60.851,-177.789,6.936,148.641
C07139=1175.122,208.065,-60.875,-177.786,6.939,148.641
C07140=1175.118,208.313,-60.899,-177.784,6.941,148.641
C07141=1175.113,208.563,-60.924,-177.781,6.943,148.641
C07142=1175.109,208.811,-60.948,-177.778,6.946,148.640
C07143=1175.104,209.060,-60.973,-177.776,6.947,148.640
C07144=1175.100,209.309,-60.998,-177.772,6.950,148.640
C07145=1175.095,209.558,-61.022,-177.770,6.952,148.640
C07146=1175.090,209.806,-61.046,-177.768,6.954,148.639
C07147=1175.086,210.077,-61.073,-177.764,6.957,148.639
C07148=1175.081,210.347,-61.100,-177.762,6.960,148.639
C07149=1175.075,210.617,-61.127,-177.759,6.961,148.639
C07150=1175.071,210.888,-61.154,-177.756,6.964,148.638
C07151=1175.067,211.137,-61.178,-177.753,6.966,148.638
C07152=1175.061,211.386,-61.203,-177.750,6.969,148.638
C07153=1175.058,211.635,-61.227,-177.748,6.971,148.637
C07154=1175.052,211.883,-61.252,-177.745,6.973,148.637
C07155=1175.048,212.132,-61.276,-177.742,6.975,148.637
C07156=1175.044,212.381,-61.301,-177.740,6.977,148.637
C07157=1175.039,212.629,-61.326,-177.737,6.979,148.637
C07158=1175.034,212.878,-61.350,-177.734,6.982,148.636
C07159=1175.030,213.127,-61.375,-177.731,6.984,148.636
C07160=1175.025,213.376,-61.399,-177.729,6.986,148.636
C07161=1175.021,213.625,-61.424,-177.726,6.988,148.636
C07162=1175.016,213.873,-61.450,-177.724,6.990,148.635
C07163=1175.012,214.121,-61.474,-177.721,6.993,148.635
C07164=1175.007,214.371,-61.499,-177.718,6.995,148.635
C07165=1175.003,214.619,-61.524,-177.716,6.997,148.635
C07166=1174.998,214.868,-61.549,-177.713,7.000,148.634
C07167=1174.993,215.117,-61.573,-177.710,7.002,148.634
C07168=1174.989,215.365,-61.597,-177.707,7.004,148.634
C07169=1174.985,215.614,-61.623,-177.705,7.006,148.634
C07170=1174.980,215.863,-61.648,-177.702,7.008,148.633
C07171=1174.976,216.112,-61.672,-177.699,7.011,148.633
C07172=1174.971,216.360,-61.698,-177.697,7.013,148.633
C07173=1174.966,216.609,-61.723,-177.694,7.015,148.633
C07174=1174.962,216.857,-61.748,-177.691,7.018,148.633
C07175=1174.958,217.107,-61.773,-177.689,7.020,148.632
C07176=1174.953,217.355,-61.797,-177.686,7.022,148.632
C07177=1174.948,217.604,-61.823,-177.683,7.024,148.632
C07178=1174.944,217.853,-61.847,-177.681,7.026,148.632
C07179=1174.940,218.101,-61.873,-177.678,7.029,148.631
C07180=1174.935,218.350,-61.898,-177.675,7.031,148.631
C07181=1174.930,218.598,-61.923,-177.672,7.034,148.631
C07182=1174.926,218.847,-61.947,-177.670,7.036,148.631
C07183=1174.922,219.096,-61.973,-177.667,7.039,148.631
C07184=1174.917,219.345,-61.998,-177.664,7.040,148.630
C07185=1174.913,219.594,-62.024,-177.662,7.042,148.630
C07186=1174.908,219.842,-62.048,-177.659,7.045,148.630
C07187=1174.904,220.091,-62.073,-177.656,7.047,148.629
C07188=1174.899,220.340,-62.098,-177.654,7.050,148.629
C07189=1174.895,220.588,-62.124,-177.651,7.052,148.629
C07190=1174.889,220.837,-62.148,-177.649,7.054,148.629
C07191=1174.885,221.086,-62.174,-177.646,7.056,148.629
C07192=1174.881,221.334,-62.199,-177.643,7.059,148.629
C07193=1174.877,221.583,-62.224,-177.640,7.061,148.628
C07194=1174.872,221.831,-62.249,-177.638,7.063,148.628
C07195=1174.867,222.081,-62.274,-177.635,7.066,148.628
C07196=1174.863,222.329,-62.300,-177.632,7.068,148.627
C07197=1174.858,222.578,-62.326,-177.630,7.070,148.627
C07198=1174.854,222.827,-62.351,-177.627,7.072,148.627
C07199=1174.849,223.075,-62.376,-177.624,7.075,148.627
C07200=1174.845,223.324,-62.401,-177.621,7.077,148.627
C07201=1174.841,223.572,-62.427,-177.619,7.079,148.627
C07202=1174.836,223.821,-62.452,-177.616,7.082,148.626
C07203=1174.832,224.070,-62.477,-177.614,7.084,148.626
C07204=1174.827,224.318,-62.503,-177.610,7.087,148.626
C07205=1174.822,224.567,-62.528,-177.608,7.089,148.626
C07206=1174.818,224.816,-62.553,-177.605,7.091,148.625
C07207=1174.813,225.064,-62.579,-177.603,7.094,148.625
C07208=1174.809,225.313,-62.605,-177.600,7.095,148.625
C07209=1174.804,225.561,-62.630,-177.597,7.098,148.625
C07210=1174.800,225.811,-62.655,-177.595,7.100,148.625
C07211=1174.796,226.060,-62.681,-177.592,7.103,148.624
C07212=1174.791,226.308,-62.706,-177.589,7.105,148.624
C07213=1174.786,226.556,-62.732,-177.587,7.108,148.624
C07214=1174.782,226.805,-62.758,-177.584,7.110,148.624
C07215=1174.777,227.053,-62.783,-177.581,7.113,148.624
C07216=1174.773,227.302,-62.809,-177.578,7.114,148.623
C07217=1174.769,227.551,-62.835,-177.576,7.117,148.623
C07218=1174.764,227.800,-62.859,-177.574,7.120,148.623
C07219=1174.760,228.048,-62.885,-177.570,7.122,148.623
C07220=1174.755,228.297,-62.911,-177.568,7.124,148.623
C07221=1174.751,228.545,-62.936,-177.565,7.127,148.622
C07222=1174.746,228.794,-62.962,-177.563,7.129,148.622
C07223=1174.741,229.043,-62.988,-177.559,7.132,148.622
C07224=1174.737,229.291,-63.014,-177.557,7.134,148.622
C07225=1174.732,229.540,-63.039,-177.554,7.136,148.622
C07226=1174.728,229.789,-63.065,-177.552,7.139,148.622
C07227=1174.724,230.038,-63.091,-177.549,7.141,148.621
C07228=1174.719,230.286,-63.116,-177.546,7.143,148.621
C07229=1174.715,230.535,-63.142,-177.544,7.145,148.621
C07230=1174.710,230.784,-63.168,-177.541,7.148,148.621
C07231=1174.705,231.031,-63.194,-177.539,7.150,148.621
C07232=1174.701,231.280,-63.220,-177.536,7.153,148.620
C07233=1174.697,231.529,-63.246,-177.533,7.155,148.620
C07234=1174.693,231.778,-63.272,-177.530,7.158,148.620
C07235=1174.688,232.026,-63.297,-177.527,7.161,148.620
C07236=1174.683,232.275,-63.323,-177.525,7.162,148.620
C07237=1174.679,232.524,-63.349,-177.522,7.165,148.619
C07238=1174.674,232.773,-63.375,-177.520,7.167,148.619
C07239=1174.671,233.021,-63.401,-177.517,7.170,148.619
C07240=1174.665,233.269,-63.427,-177.514,7.172,148.619
C07241=1174.661,233.518,-63.453,-177.511,7.175,148.619
C07242=1174.657,233.767,-63.479,-177.509,7.177,148.619
C07243=1174.652,234.016,-63.505,-177.506,7.180,148.618
C07244=1174.648,234.264,-63.532,-177.504,7.182,148.618
C07245=1174.643,234.512,-63.557,-177.501,7.185,148.618
C07246=1174.639,234.761,-63.583,-177.498,7.187,148.618
C07247=1174.634,235.010,-63.609,-177.496,7.190,148.618
C07248=1174.630,235.258,-63.636,-177.493,7.191,148.617
C07249=1174.625,235.507,-63.661,-177.490,7.194,148.617
C07250=1174.621,235.755,-63.687,-177.488,7.196,148.617
C07251=1174.616,236.027,-63.716,-177.485,7.199,148.617
C07252=1174.611,236.299,-63.744,-177.482,7.202,148.617
C07253=1174.606,236.570,-63.773,-177.479,7.205,148.616
C07254=1174.601,236.842,-63.802,-177.476,7.208,148.616
C07255=1174.597,237.090,-63.828,-177.473,7.209,148.616
C07256=1174.593,237.339,-63.854,-177.471,7.212,148.616
C07257=1174.588,237.588,-63.881,-177.468,7.214,148.616
C07258=1174.583,237.836,-63.906,-177.465,7.217,148.616
C07259=1174.578,238.085,-63.933,-177.462,7.220,148.616
C07260=1174.575,238.333,-63.959,-177.460,7.222,148.615
C07261=1174.570,238.582,-63.985,-177.457,7.225,148.615
C07262=1174.566,238.830,-64.012,-177.455,7.227,148.615
C07263=1174.561,239.079,-64.038,-177.452,7.230,148.615
C07264=1174.557,239.328,-64.065,-177.449,7.232,148.615
C07265=1174.553,239.576,-64.090,-177.447,7.235,148.615
C07266=1174.548,239.825,-64.117,-177.444,7.237,148.614
C07267=1174.544,240.074,-64.143,-177.441,7.239,148.614
C07268=1174.539,240.322,-64.170,-177.439,7.242,148.614
C07269=1174.534,240.570,-64.196,-177.436,7.244,148.614
C07270=1174.530,240.819,-64.222,-177.433,7.247,148.614
C07271=1174.525,241.068,-64.248,-177.431,7.249,148.614
C07272=1174.521,241.316,-64.275,-177.428,7.252,148.613
C07273=1174.517,241.564,-64.302,-177.426,7.254,148.613
C07274=1174.512,241.813,-64.328,-177.423,7.257,148.613
C07275=1174.508,242.062,-64.355,-177.420,7.260,148.613
C07276=1174.503,242.310,-64.382,-177.417,7.262,148.613
C07277=1174.499,242.559,-64.408,-177.415,7.265,148.613
C07278=1174.494,242.807,-64.435,-177.412,7.267,148.612
C07279=1174.490,243.056,-64.461,-177.409,7.270,148.612
C07280=1174.485,243.305,-64.487,-177.406,7.273,148.612
C07281=1174.481,243.553,-64.514,-177.404,7.274,148.612
C07282=1174.477,243.801,-64.541,-177.401,7.277,148.612
C07283=1174.473,244.050,-64.567,-177.399,7.279,148.612
C07284=1174.468,244.299,-64.594,-177.396,7.282,148.612
C07285=1174.463,244.547,-64.621,-177.393,7.285,148.611
C07286=1174.459,244.795,-64.647,-177.391,7.287,148.611
C07287=1174.454,245.045,-64.674,-177.388,7.290,148.611
C07288=1174.450,245.293,-64.701,-177.385,7.292,148.611
C07289=1174.446,245.541,-64.727,-177.383,7.295,148.611
C07290=1174.441,245.790,-64.754,-177.380,7.298,148.611
C07291=1174.437,246.038,-64.781,-177.378,7.300,148.611
C07292=1174.433,246.286,-64.808,-177.374,7.303,148.610
C07293=1174.428,246.535,-64.834,-177.372,7.305,148.610
C07294=1174.424,246.784,-64.861,-177.370,7.308,148.610
C07295=1174.420,247.033,-64.888,-177.366,7.310,148.610
C07296=1174.415,247.281,-64.915,-177.364,7.313,148.610
C07297=1174.410,247.530,-64.942,-177.361,7.316,148.610
C07298=1174.406,247.778,-64.969,-177.359,7.318,148.610
C07299=1174.402,248.027,-64.996,-177.356,7.320,148.609
C07300=1174.397,248.275,-65.023,-177.353,7.323,148.609
C07301=1174.392,248.524,-65.050,-177.351,7.325,148.609
C07302=1174.389,248.772,-65.076,-177.348,7.328,148.609
C07303=1174.384,249.020,-65.103,-177.345,7.331,148.609
C07304=1174.379,249.269,-65.130,-177.343,7.333,148.609
C07305=1174.375,249.517,-65.157,-177.340,7.336,148.609
C07306=1174.371,249.766,-65.184,-177.337,7.339,148.609
C07307=1174.367,250.015,-65.211,-177.335,7.341,148.608
C07308=1174.362,250.263,-65.238,-177.332,7.344,148.608
C07309=1174.357,250.512,-65.265,-177.330,7.346,148.608
C07310=1174.353,250.760,-65.293,-177.327,7.349,148.608
C07311=1174.349,251.008,-65.319,-177.324,7.352,148.608
C07312=1174.344,251.257,-65.346,-177.322,7.354,148.608
C07313=1174.340,251.506,-65.374,-177.319,7.357,148.608
C07314=1174.335,251.754,-65.401,-177.316,7.360,148.608
C07315=1174.331,252.003,-65.428,-177.314,7.362,148.608
C07316=1174.326,252.251,-65.455,-177.311,7.364,148.607
C07317=1174.322,252.499,-65.482,-177.308,7.367,148.607
C07318=1174.318,252.747,-65.509,-177.306,7.370,148.607
C07319=1174.314,252.997,-65.536,-177.303,7.373,148.607
C07320=1174.309,253.245,-65.563,-177.300,7.376,148.607
C07321=1174.304,253.494,-65.590,-177.298,7.377,148.607
C07322=1174.300,253.742,-65.618,-177.295,7.380,148.607
C07323=1174.295,253.990,-65.645,-177.292,7.383,148.607
C07324=1174.291,254.239,-65.673,-177.290,7.385,148.607
C07325=1174.287,254.488,-65.700,-177.287,7.388,148.606
